LIN {X 0,Y 235.137,Z 262.859,A -85,B 0,C 180,E1 -19747.889,E2 -19747.889} C_VEL
LIN {X 0,Y 235.031,Z 260.731,A -85,B 0,C 180,E1 -19751.62,E2 -19751.62} C_VEL
LIN {X 0,Y 234.887,Z 259.391,A -85,B 0,C 180,E1 -19754.102,E2 -19754.102} C_VEL
LIN {X 0,Y 234.882,Z 259.229,A -85,B 0,C 180,E1 -19758.416,E2 -19758.416} C_VEL
LIN {X 0,Y 234.948,Z 259.217,A -85,B 0,C 180,E1 -19761.084,E2 -19761.084} C_VEL
LIN {X 0,Y 234.953,Z 259.217,A -85,B 0,C 180,E1 -19765.365,E2 -19765.365} C_VEL
LIN {X 0,Y 234.961,Z 259.216,A -85,B 0,C 180,E1 -19770.156,E2 -19770.156} C_VEL
LIN {X 0,Y 234.985,Z 259.213,A -85,B 0,C 180,E1 -19773.792,E2 -19773.792} C_VEL
LIN {X 0,Y 235.002,Z 259.213,A -85,B 0,C 180,E1 -19778.969,E2 -19778.969} C_VEL
LIN {X 0,Y 235.086,Z 259.202,A -85,B 0,C 180,E1 -19783.058,E2 -19783.058} C_VEL
LIN {X 0,Y 235.136,Z 259.195,A -85,B 0,C 180,E1 -19787.923,E2 -19787.923} C_VEL
LIN {X 0,Y 235.381,Z 259.165,A -85,B 0,C 180,E1 -19791.414,E2 -19791.414} C_VEL
LIN {X 0,Y 235.397,Z 259.162,A -85,B 0,C 180,E1 -19793.141,E2 -19793.141} C_VEL
LIN {X 0,Y 235.593,Z 259.138,A -85,B 0,C 180,E1 -19798.29,E2 -19798.29} C_VEL
LIN {X 0,Y 235.586,Z 259.141,A -85,B 0,C 180,E1 -19801.709,E2 -19801.709} C_VEL
LIN {X 0,Y 235.397,Z 259.162,A -85,B 0,C 180,E1 -19806.859,E2 -19806.859} C_VEL
LIN {X 0,Y 235.243,Z 259.182,A -85,B 0,C 180,E1 -19810.326,E2 -19810.326} C_VEL
LIN {X 0,Y 235.103,Z 259.191,A -85,B 0,C 180,E1 -19815.607,E2 -19815.607} C_VEL
LIN {X 0,Y 234.998,Z 259.206,A -85,B 0,C 180,E1 -19819.206,E2 -19819.206} C_VEL
LIN {X 0,Y 234.951,Z 259.218,A -85,B 0,C 180,E1 -19822.884,E2 -19822.884} C_VEL
LIN {X 0,Y 234.96,Z 259.218,A -85,B 0,C 180,E1 -19826.658,E2 -19826.658} C_VEL
LIN {X 0,Y 235.019,Z 259.356,A -85,B 0,C 180,E1 -19829.456,E2 -19829.456} C_VEL
LIN {X 0,Y 235.474,Z 262.099,A -85,B 0,C 180,E1 -19833.317,E2 -19833.317} C_VEL
LIN {X 0,Y 235.891,Z 264.612,A -85,B 0,C 180,E1 -19836.574,E2 -19836.574} C_VEL
LIN {X 0,Y 236.478,Z 268.222,A -85,B 0,C 180,E1 -19840.831,E2 -19840.831} C_VEL
LIN {X 0,Y 237.176,Z 271.785,A -85,B 0,C 180,E1 -19844.674,E2 -19844.674} C_VEL
LIN {X 0,Y 237.723,Z 274.689,A -85,B 0,C 180,E1 -19847.655,E2 -19847.655} C_VEL
LIN {X 0,Y 238.213,Z 278.061,A -85,B 0,C 180,E1 -19850.898,E2 -19850.898} C_VEL
LIN {X 0,Y 237.534,Z 279.156,A -85,B 0,C 180,E1 -19851.795,E2 -19851.795} C_VEL
LIN {X 0,Y 234.488,Z 281.133,A -85,B 0,C 180,E1 -19853.167,E2 -19853.167} C_VEL
LIN {X 0,Y 231.288,Z 283.125,A -85,B 0,C 180,E1 -19854.569,E2 -19854.569} C_VEL
LIN {X 0,Y 230.426,Z 284.271,A -85,B 0,C 180,E1 -19855.504,E2 -19855.504} C_VEL
LIN {X 0,Y 230.39,Z 284.412,A -85,B 0,C 180,E1 -19855.627,E2 -19855.627} C_VEL
LIN {X 0,Y 231.203,Z 287.728,A -85,B 0,C 180,E1 -19855.945,E2 -19855.945} C_VEL
LIN {X 0,Y 234.78,Z 300.694,A -85,B 0,C 180,E1 -19857.465,E2 -19857.465} C_VEL
LIN {X 0,Y 237.057,Z 312.469,A -85,B 0,C 180,E1 -19858.986,E2 -19858.986} C_VEL
LIN {X 0,Y 238.455,Z 324.771,A -85,B 0,C 180,E1 -19860.767,E2 -19860.767} C_VEL
LIN {X 0,Y 238.796,Z 335.33,A -85,B 0,C 180,E1 -19862.512,E2 -19862.512} C_VEL
LIN {X 0,Y 238.284,Z 345.559,A -85,B 0,C 180,E1 -19864.45,E2 -19864.45} C_VEL
LIN {X 0,Y 236.518,Z 352.666,A -85,B 0,C 180,E1 -19865.888,E2 -19865.888} C_VEL
LIN {X 0,Y 234.021,Z 361.179,A -85,B 0,C 180,E1 -19867.954,E2 -19867.954} C_VEL
LIN {X 0,Y 231.65,Z 369.503,A -85,B 0,C 180,E1 -19870.508,E2 -19870.508} C_VEL
LIN {X 0,Y 229.654,Z 376.233,A -85,B 0,C 180,E1 -19873.102,E2 -19873.102} C_VEL
LIN {X 0,Y 227.937,Z 381.62,A -85,B 0,C 180,E1 -19875.723,E2 -19875.723} C_VEL
LIN {X 0,Y 226.866,Z 385.849,A -85,B 0,C 180,E1 -19878.386,E2 -19878.386} C_VEL
LIN {X 0,Y 226.17,Z 389.027,A -85,B 0,C 180,E1 -19881.064,E2 -19881.064} C_VEL
LIN {X 0,Y 225.931,Z 390.624,A -85,B 0,C 180,E1 -19882.855,E2 -19882.855} C_VEL
LIN {X 0,Y 225.839,Z 391.843,A -85,B 0,C 180,E1 -19884.763,E2 -19884.763} C_VEL
LIN {X 0,Y 225.885,Z 392.883,A -85,B 0,C 180,E1 -19888.22,E2 -19888.22} C_VEL
LIN {X 0,Y 225.95,Z 392.842,A -85,B 0,C 180,E1 -19890.003,E2 -19890.003} C_VEL
LIN {X 0,Y 225.909,Z 392.378,A -85,B 0,C 180,E1 -19891.785,E2 -19891.785} C_VEL
LIN {X 0,Y 225.864,Z 391.475,A -85,B 0,C 180,E1 -19893.571,E2 -19893.571} C_VEL
LIN {X 0,Y 225.883,Z 390.17,A -85,B 0,C 180,E1 -19895.358,E2 -19895.358} C_VEL
LIN {X 0,Y 226.081,Z 387.399,A -85,B 0,C 180,E1 -19898.044,E2 -19898.044} C_VEL
LIN {X 0,Y 226.596,Z 383.592,A -85,B 0,C 180,E1 -19900.727,E2 -19900.727} C_VEL
LIN {X 0,Y 227.465,Z 378.65,A -85,B 0,C 180,E1 -19903.401,E2 -19903.401} C_VEL
LIN {X 0,Y 228.927,Z 372.442,A -85,B 0,C 180,E1 -19906.042,E2 -19906.042} C_VEL
LIN {X 0,Y 230.66,Z 364.83,A -85,B 0,C 180,E1 -19908.623,E2 -19908.623} C_VEL
LIN {X 0,Y 232.391,Z 356.97,A -85,B 0,C 180,E1 -19910.771,E2 -19910.771} C_VEL
LIN {X 0,Y 234.323,Z 348.211,A -85,B 0,C 180,E1 -19912.718,E2 -19912.718} C_VEL
LIN {X 0,Y 235.388,Z 342.642,A -85,B 0,C 180,E1 -19913.773,E2 -19913.773} C_VEL
LIN {X 0,Y 235.357,Z 331.167,A -85,B 0,C 180,E1 -19915.788,E2 -19915.788} C_VEL
LIN {X 0,Y 234.896,Z 319.818,A -85,B 0,C 180,E1 -19917.434,E2 -19917.434} C_VEL
LIN {X 0,Y 233.577,Z 307.331,A -85,B 0,C 180,E1 -19918.943,E2 -19918.943} C_VEL
LIN {X 0,Y 231.149,Z 294.067,A -85,B 0,C 180,E1 -19920.296,E2 -19920.296} C_VEL
LIN {X 0,Y 229.071,Z 284.971,A -85,B 0,C 180,E1 -19921.1,E2 -19921.1} C_VEL
LIN {X 0,Y 230.358,Z 279.833,A -85,B 0,C 180,E1 -19925.43,E2 -19925.43} C_VEL
LIN {X 0,Y 230.728,Z 277.284,A -85,B 0,C 180,E1 -19927.631,E2 -19927.631} C_VEL
LIN {X 0,Y 230.496,Z 274.331,A -85,B 0,C 180,E1 -19930.335,E2 -19930.335} C_VEL
LIN {X 0,Y 229.629,Z 269.831,A -85,B 0,C 180,E1 -19934.747,E2 -19934.747} C_VEL
LIN {X 0,Y 228.975,Z 266.081,A -85,B 0,C 180,E1 -19938.707,E2 -19938.707} C_VEL
LIN {X 0,Y 228.326,Z 262.168,A -85,B 0,C 180,E1 -19943.162,E2 -19943.162} C_VEL
LIN {X 0,Y 227.892,Z 260.098,A -85,B 0,C 180,E1 -19945.749,E2 -19945.749} C_VEL
LIN {X 0,Y 227.884,Z 260.098,A -85,B 0,C 180,E1 -19950.433,E2 -19950.433} C_VEL
LIN {X 0,Y 227.912,Z 260.095,A -85,B 0,C 180,E1 -19954.424,E2 -19954.424} C_VEL
LIN {X 0,Y 227.955,Z 260.091,A -85,B 0,C 180,E1 -19958.286,E2 -19958.286} C_VEL
LIN {X 0,Y 227.998,Z 260.084,A -85,B 0,C 180,E1 -19962.864,E2 -19962.864} C_VEL
LIN {X 0,Y 228.051,Z 260.08,A -85,B 0,C 180,E1 -19967.542,E2 -19967.542} C_VEL
LIN {X 0,Y 228.259,Z 260.053,A -85,B 0,C 180,E1 -19971.144,E2 -19971.144} C_VEL
LIN {X 0,Y 228.325,Z 260.041,A -85,B 0,C 180,E1 -19972.928,E2 -19972.928} C_VEL
LIN {X 0,Y 228.562,Z 260.014,A -85,B 0,C 180,E1 -19978.238,E2 -19978.238} C_VEL
LIN {X 0,Y 228.547,Z 260.017,A -85,B 0,C 180,E1 -19981.762,E2 -19981.762} C_VEL
LIN {X 0,Y 228.309,Z 260.046,A -85,B 0,C 180,E1 -19987.073,E2 -19987.073} C_VEL
LIN {X 0,Y 228.151,Z 260.061,A -85,B 0,C 180,E1 -19990.651,E2 -19990.651} C_VEL
LIN {X 0,Y 228.046,Z 260.074,A -85,B 0,C 180,E1 -19994.274,E2 -19994.274} C_VEL
LIN {X 0,Y 227.962,Z 260.087,A -85,B 0,C 180,E1 -19997.957,E2 -19997.957} C_VEL
LIN {X 0,Y 227.913,Z 260.095,A -85,B 0,C 180,E1 -20002.312,E2 -20002.312} C_VEL
LIN {X 0,Y 227.91,Z 260.096,A -85,B 0,C 180,E1 -20006.581,E2 -20006.581} C_VEL
LIN {X 0,Y 227.878,Z 260.098,A -85,B 0,C 180,E1 -20010.278,E2 -20010.278} C_VEL
LIN {X 0,Y 227.885,Z 260.095,A -85,B 0,C 180,E1 -20013.72,E2 -20013.72} C_VEL
LIN {X 0,Y 227.852,Z 260.102,A -85,B 0,C 180,E1 -20018.09,E2 -20018.09} C_VEL
LIN {X 0,Y 227.813,Z 260.106,A -85,B 0,C 180,E1 -20022.742,E2 -20022.742} C_VEL
LIN {X 0,Y 227.797,Z 260.109,A -85,B 0,C 180,E1 -20027.251,E2 -20027.251} C_VEL
LIN {X 0,Y 227.844,Z 260.104,A -85,B 0,C 180,E1 -20031.906,E2 -20031.906} C_VEL
LIN {X 0,Y 227.82,Z 260.105,A -85,B 0,C 180,E1 -20036.267,E2 -20036.267} C_VEL
LIN {X 0,Y 227.682,Z 260.118,A -85,B 0,C 180,E1 -20038.346,E2 -20038.346} C_VEL
LIN {X 0,Y 227.603,Z 260.825,A -85,B 0,C 180,E1 -20040.39,E2 -20040.39} C_VEL
LIN {X 0,Y 227.534,Z 262.75,A -85,B 0,C 180,E1 -20043.143,E2 -20043.143} C_VEL
LIN {X 0,Y 228.668,Z 265.801,A -85,B 0,C 180,E1 -20043.474,E2 -20043.474} C_VEL
LIN {X 0,Y 232.897,Z 277.354,A -85,B 0,C 180,E1 -20044.864,E2 -20044.864} C_VEL
LIN {X 0,Y 235.978,Z 288.099,A -85,B 0,C 180,E1 -20046.305,E2 -20046.305} C_VEL
LIN {X 0,Y 238.279,Z 299.414,A -85,B 0,C 180,E1 -20048.005,E2 -20048.005} C_VEL
LIN {X 0,Y 239.076,Z 305.229,A -85,B 0,C 180,E1 -20048.976,E2 -20048.976} C_VEL
LIN {X 0,Y 237.375,Z 315.143,A -85,B 0,C 180,E1 -20050.542,E2 -20050.542} C_VEL
LIN {X 0,Y 235.171,Z 325.68,A -85,B 0,C 180,E1 -20052.609,E2 -20052.609} C_VEL
LIN {X 0,Y 233.368,Z 333.508,A -85,B 0,C 180,E1 -20054.516,E2 -20054.516} C_VEL
LIN {X 0,Y 231.558,Z 341.294,A -85,B 0,C 180,E1 -20056.84,E2 -20056.84} C_VEL
LIN {X 0,Y 229.715,Z 348.233,A -85,B 0,C 180,E1 -20059.42,E2 -20059.42} C_VEL
LIN {X 0,Y 228.841,Z 352.047,A -85,B 0,C 180,E1 -20061.164,E2 -20061.164} C_VEL
LIN {X 0,Y 227.754,Z 356.785,A -85,B 0,C 180,E1 -20063.797,E2 -20063.797} C_VEL
LIN {X 0,Y 226.813,Z 360.44,A -85,B 0,C 180,E1 -20066.444,E2 -20066.444} C_VEL
LIN {X 0,Y 226.45,Z 362.325,A -85,B 0,C 180,E1 -20068.219,E2 -20068.219} C_VEL
LIN {X 0,Y 226.197,Z 363.78,A -85,B 0,C 180,E1 -20069.997,E2 -20069.997} C_VEL
LIN {X 0,Y 226.135,Z 365.446,A -85,B 0,C 180,E1 -20073.561,E2 -20073.561} C_VEL
LIN {X 0,Y 226.283,Z 365.678,A -85,B 0,C 180,E1 -20076.342,E2 -20076.342} C_VEL
LIN {X 0,Y 226.504,Z 365.058,A -85,B 0,C 180,E1 -20078.922,E2 -20078.922} C_VEL
LIN {X 0,Y 227.34,Z 362.821,A -85,B 0,C 180,E1 -20082.495,E2 -20082.495} C_VEL
LIN {X 0,Y 228.402,Z 360.02,A -85,B 0,C 180,E1 -20085.159,E2 -20085.159} C_VEL
LIN {X 0,Y 229.798,Z 356.193,A -85,B 0,C 180,E1 -20087.806,E2 -20087.806} C_VEL
LIN {X 0,Y 231.579,Z 351.225,A -85,B 0,C 180,E1 -20090.424,E2 -20090.424} C_VEL
LIN {X 0,Y 233.827,Z 344.95,A -85,B 0,C 180,E1 -20092.997,E2 -20092.997} C_VEL
LIN {X 0,Y 236.355,Z 337.063,A -85,B 0,C 180,E1 -20095.538,E2 -20095.538} C_VEL
LIN {X 0,Y 238.723,Z 329.001,A -85,B 0,C 180,E1 -20097.622,E2 -20097.622} C_VEL
LIN {X 0,Y 241.366,Z 319.137,A -85,B 0,C 180,E1 -20099.667,E2 -20099.667} C_VEL
LIN {X 0,Y 243.113,Z 311.993,A -85,B 0,C 180,E1 -20100.869,E2 -20100.869} C_VEL
LIN {X 0,Y 241.935,Z 302.961,A -85,B 0,C 180,E1 -20102.602,E2 -20102.602} C_VEL
LIN {X 0,Y 239.585,Z 292.859,A -85,B 0,C 180,E1 -20104.409,E2 -20104.409} C_VEL
LIN {X 0,Y 235.756,Z 280.778,A -85,B 0,C 180,E1 -20106.4,E2 -20106.4} C_VEL
LIN {X 0,Y 231.266,Z 270.388,A -85,B 0,C 180,E1 -20108.062,E2 -20108.062} C_VEL
LIN {X 0,Y 229.347,Z 266.528,A -85,B 0,C 180,E1 -20108.669,E2 -20108.669} C_VEL
LIN {X 0,Y 228.101,Z 263.373,A -85,B 0,C 180,E1 -20109.132,E2 -20109.132} C_VEL
LIN {X 0,Y 227.97,Z 261.447,A -85,B 0,C 180,E1 -20112.702,E2 -20112.702} C_VEL
LIN {X 0,Y 227.819,Z 260.161,A -85,B 0,C 180,E1 -20115.192,E2 -20115.192} C_VEL
LIN {X 0,Y 227.825,Z 260.106,A -85,B 0,C 180,E1 -20119.623,E2 -20119.623} C_VEL
LIN {X 0,Y 227.892,Z 260.096,A -85,B 0,C 180,E1 -20124.13,E2 -20124.13} C_VEL
LIN {X 0,Y 227.864,Z 260.099,A -85,B 0,C 180,E1 -20128.376,E2 -20128.376} C_VEL
LIN {X 0,Y 227.877,Z 260.093,A -85,B 0,C 180,E1 -20132.443,E2 -20132.443} C_VEL
LIN {X 0,Y 227.905,Z 260.097,A -85,B 0,C 180,E1 -20136.366,E2 -20136.366} C_VEL
LIN {X 0,Y 227.933,Z 260.092,A -85,B 0,C 180,E1 -20140.173,E2 -20140.173} C_VEL
LIN {X 0,Y 228.048,Z 260.077,A -85,B 0,C 180,E1 -20143.897,E2 -20143.897} C_VEL
LIN {X 0,Y 228.161,Z 260.066,A -85,B 0,C 180,E1 -20149.349,E2 -20149.349} C_VEL
LIN {X 0,Y 228.349,Z 260.04,A -85,B 0,C 180,E1 -20152.928,E2 -20152.928} C_VEL
LIN {X 0,Y 228.553,Z 260.015,A -85,B 0,C 180,E1 -20158.238,E2 -20158.238} C_VEL
LIN {X 0,Y 228.545,Z 260.018,A -85,B 0,C 180,E1 -20161.762,E2 -20161.762} C_VEL
LIN {X 0,Y 228.349,Z 260.04,A -85,B 0,C 180,E1 -20167.071,E2 -20167.071} C_VEL
LIN {X 0,Y 228.161,Z 260.063,A -85,B 0,C 180,E1 -20170.65,E2 -20170.65} C_VEL
LIN {X 0,Y 228.047,Z 260.071,A -85,B 0,C 180,E1 -20176.103,E2 -20176.103} C_VEL
LIN {X 0,Y 227.932,Z 260.088,A -85,B 0,C 180,E1 -20179.826,E2 -20179.826} C_VEL
LIN {X 0,Y 227.904,Z 260.098,A -85,B 0,C 180,E1 -20183.634,E2 -20183.634} C_VEL
LIN {X 0,Y 227.891,Z 260.132,A -85,B 0,C 180,E1 -20188.054,E2 -20188.054} C_VEL
LIN {X 0,Y 228.311,Z 262.418,A -85,B 0,C 180,E1 -20191.554,E2 -20191.554} C_VEL
LIN {X 0,Y 228.812,Z 265.456,A -85,B 0,C 180,E1 -20195.703,E2 -20195.703} C_VEL
LIN {X 0,Y 229.4,Z 268.969,A -85,B 0,C 180,E1 -20200.043,E2 -20200.043} C_VEL
LIN {X 0,Y 229.887,Z 271.346,A -85,B 0,C 180,E1 -20202.805,E2 -20202.805} C_VEL
LIN {X 0,Y 230.615,Z 275.277,A -85,B 0,C 180,E1 -20207.004,E2 -20207.004} C_VEL
LIN {X 0,Y 231.178,Z 278.574,A -85,B 0,C 180,E1 -20210.33,E2 -20210.33} C_VEL
LIN {X 0,Y 231.238,Z 280.951,A -85,B 0,C 180,E1 -20212.569,E2 -20212.569} C_VEL
LIN {X 0,Y 230.426,Z 284.271,A -85,B 0,C 180,E1 -20215.504,E2 -20215.504} C_VEL
LIN {X 0,Y 231.228,Z 285.071,A -85,B 0,C 180,E1 -20215.808,E2 -20215.808} C_VEL
LIN {X 0,Y 233.342,Z 287.602,A -85,B 0,C 180,E1 -20216.31,E2 -20216.31} C_VEL
LIN {X 0,Y 234.902,Z 290.926,A -85,B 0,C 180,E1 -20216.743,E2 -20216.743} C_VEL
LIN {X 0,Y 235.443,Z 294.756,A -85,B 0,C 180,E1 -20217.111,E2 -20217.111} C_VEL
LIN {X 0,Y 235.158,Z 299.092,A -85,B 0,C 180,E1 -20217.313,E2 -20217.313} C_VEL
LIN {X 0,Y 232.838,Z 305.681,A -85,B 0,C 180,E1 -20217.51,E2 -20217.51} C_VEL
LIN {X 0,Y 230.998,Z 310.912,A -85,B 0,C 180,E1 -20217.847,E2 -20217.847} C_VEL
LIN {X 0,Y 230.809,Z 313.949,A -85,B 0,C 180,E1 -20218.202,E2 -20218.202} C_VEL
LIN {X 0,Y 232.06,Z 326.581,A -85,B 0,C 180,E1 -20220.164,E2 -20220.164} C_VEL
LIN {X 0,Y 232.24,Z 337.478,A -85,B 0,C 180,E1 -20222.09,E2 -20222.09} C_VEL
LIN {X 0,Y 231.473,Z 347.568,A -85,B 0,C 180,E1 -20224.125,E2 -20224.125} C_VEL
LIN {X 0,Y 228.928,Z 356.07,A -85,B 0,C 180,E1 -20226.001,E2 -20226.001} C_VEL
LIN {X 0,Y 226.109,Z 365.279,A -85,B 0,C 180,E1 -20228.57,E2 -20228.57} C_VEL
LIN {X 0,Y 223.823,Z 372.77,A -85,B 0,C 180,E1 -20231.228,E2 -20231.228} C_VEL
LIN {X 0,Y 221.593,Z 379.667,A -85,B 0,C 180,E1 -20234.363,E2 -20234.363} C_VEL
LIN {X 0,Y 220.177,Z 384.236,A -85,B 0,C 180,E1 -20237.092,E2 -20237.092} C_VEL
LIN {X 0,Y 219.588,Z 386.662,A -85,B 0,C 180,E1 -20238.931,E2 -20238.931} C_VEL
LIN {X 0,Y 219.137,Z 388.658,A -85,B 0,C 180,E1 -20240.775,E2 -20240.775} C_VEL
LIN {X 0,Y 218.856,Z 390.243,A -85,B 0,C 180,E1 -20242.623,E2 -20242.623} C_VEL
LIN {X 0,Y 218.74,Z 391.573,A -85,B 0,C 180,E1 -20244.884,E2 -20244.884} C_VEL
LIN {X 0,Y 218.815,Z 392.462,A -85,B 0,C 180,E1 -20248.162,E2 -20248.162} C_VEL
LIN {X 0,Y 218.878,Z 392.411,A -85,B 0,C 180,E1 -20250.003,E2 -20250.003} C_VEL
LIN {X 0,Y 218.838,Z 391.925,A -85,B 0,C 180,E1 -20251.843,E2 -20251.843} C_VEL
LIN {X 0,Y 218.784,Z 389.925,A -85,B 0,C 180,E1 -20255.244,E2 -20255.244} C_VEL
LIN {X 0,Y 219.043,Z 386.899,A -85,B 0,C 180,E1 -20258.304,E2 -20258.304} C_VEL
LIN {X 0,Y 219.596,Z 383.067,A -85,B 0,C 180,E1 -20261.074,E2 -20261.074} C_VEL
LIN {X 0,Y 220.533,Z 378.098,A -85,B 0,C 180,E1 -20263.831,E2 -20263.831} C_VEL
LIN {X 0,Y 222.031,Z 371.857,A -85,B 0,C 180,E1 -20266.554,E2 -20266.554} C_VEL
LIN {X 0,Y 223.782,Z 364.6,A -85,B 0,C 180,E1 -20269.085,E2 -20269.085} C_VEL
LIN {X 0,Y 225.736,Z 356.116,A -85,B 0,C 180,E1 -20271.461,E2 -20271.461} C_VEL
LIN {X 0,Y 227.976,Z 346.407,A -85,B 0,C 180,E1 -20273.628,E2 -20273.628} C_VEL
LIN {X 0,Y 228.546,Z 343.068,A -85,B 0,C 180,E1 -20274.289,E2 -20274.289} C_VEL
LIN {X 0,Y 228.641,Z 330.99,A -85,B 0,C 180,E1 -20276.49,E2 -20276.49} C_VEL
LIN {X 0,Y 228.27,Z 320.835,A -85,B 0,C 180,E1 -20278.033,E2 -20278.033} C_VEL
LIN {X 0,Y 226.993,Z 307.895,A -85,B 0,C 180,E1 -20279.698,E2 -20279.698} C_VEL
LIN {X 0,Y 224.528,Z 294.296,A -85,B 0,C 180,E1 -20281.164,E2 -20281.164} C_VEL
LIN {X 0,Y 222.295,Z 285.273,A -85,B 0,C 180,E1 -20282.009,E2 -20282.009} C_VEL
LIN {X 0,Y 222.241,Z 284.55,A -85,B 0,C 180,E1 -20282.072,E2 -20282.072} C_VEL
LIN {X 0,Y 223.143,Z 281.169,A -85,B 0,C 180,E1 -20285.027,E2 -20285.027} C_VEL
LIN {X 0,Y 223.579,Z 279.31,A -85,B 0,C 180,E1 -20286.676,E2 -20286.676} C_VEL
LIN {X 0,Y 223.665,Z 276.847,A -85,B 0,C 180,E1 -20288.938,E2 -20288.938} C_VEL
LIN {X 0,Y 223.07,Z 273.235,A -85,B 0,C 180,E1 -20292.46,E2 -20292.46} C_VEL
LIN {X 0,Y 222.319,Z 269.265,A -85,B 0,C 180,E1 -20296.646,E2 -20296.646} C_VEL
LIN {X 0,Y 221.662,Z 265.72,A -85,B 0,C 180,E1 -20300.645,E2 -20300.645} C_VEL
LIN {X 0,Y 221.405,Z 263.799,A -85,B 0,C 180,E1 -20302.907,E2 -20302.907} C_VEL
LIN {X 0,Y 220.845,Z 260.976,A -85,B 0,C 180,E1 -20306.521,E2 -20306.521} C_VEL
LIN {X 0,Y 220.842,Z 260.975,A -85,B 0,C 180,E1 -20309.391,E2 -20309.391} C_VEL
LIN {X 0,Y 220.884,Z 260.969,A -85,B 0,C 180,E1 -20313.548,E2 -20313.548} C_VEL
LIN {X 0,Y 220.877,Z 260.971,A -85,B 0,C 180,E1 -20317.553,E2 -20317.553} C_VEL
LIN {X 0,Y 220.936,Z 260.965,A -85,B 0,C 180,E1 -20322.62,E2 -20322.62} C_VEL
LIN {X 0,Y 220.984,Z 260.959,A -85,B 0,C 180,E1 -20327.137,E2 -20327.137} C_VEL
LIN {X 0,Y 221.196,Z 260.932,A -85,B 0,C 180,E1 -20330.859,E2 -20330.859} C_VEL
LIN {X 0,Y 221.259,Z 260.921,A -85,B 0,C 180,E1 -20332.701,E2 -20332.701} C_VEL
LIN {X 0,Y 221.52,Z 260.891,A -85,B 0,C 180,E1 -20338.182,E2 -20338.182} C_VEL
LIN {X 0,Y 221.481,Z 260.897,A -85,B 0,C 180,E1 -20341.819,E2 -20341.819} C_VEL
LIN {X 0,Y 221.247,Z 260.927,A -85,B 0,C 180,E1 -20347.3,E2 -20347.3} C_VEL
LIN {X 0,Y 221.072,Z 260.945,A -85,B 0,C 180,E1 -20350.996,E2 -20350.996} C_VEL
LIN {X 0,Y 220.988,Z 260.957,A -85,B 0,C 180,E1 -20356.632,E2 -20356.632} C_VEL
LIN {X 0,Y 220.883,Z 260.966,A -85,B 0,C 180,E1 -20360.487,E2 -20360.487} C_VEL
LIN {X 0,Y 220.806,Z 260.977,A -85,B 0,C 180,E1 -20364.443,E2 -20364.443} C_VEL
LIN {X 0,Y 220.804,Z 260.979,A -85,B 0,C 180,E1 -20368.519,E2 -20368.519} C_VEL
LIN {X 0,Y 220.82,Z 260.976,A -85,B 0,C 180,E1 -20372.756,E2 -20372.756} C_VEL
LIN {X 0,Y 220.819,Z 260.977,A -85,B 0,C 180,E1 -20377.277,E2 -20377.277} C_VEL
LIN {X 0,Y 220.803,Z 260.98,A -85,B 0,C 180,E1 -20380.187,E2 -20380.187} C_VEL
LIN {X 0,Y 220.773,Z 260.985,A -85,B 0,C 180,E1 -20384.455,E2 -20384.455} C_VEL
LIN {X 0,Y 220.756,Z 260.987,A -85,B 0,C 180,E1 -20388.041,E2 -20388.041} C_VEL
LIN {X 0,Y 220.832,Z 260.977,A -85,B 0,C 180,E1 -20392.791,E2 -20392.791} C_VEL
LIN {X 0,Y 220.693,Z 260.991,A -85,B 0,C 180,E1 -20397.22,E2 -20397.22} C_VEL
LIN {X 0,Y 220.612,Z 261.328,A -85,B 0,C 180,E1 -20399.353,E2 -20399.353} C_VEL
LIN {X 0,Y 220.493,Z 263.082,A -85,B 0,C 180,E1 -20402.107,E2 -20402.107} C_VEL
LIN {X 0,Y 221.673,Z 266.22,A -85,B 0,C 180,E1 -20402.467,E2 -20402.467} C_VEL
LIN {X 0,Y 225.988,Z 277.513,A -85,B 0,C 180,E1 -20403.922,E2 -20403.922} C_VEL
LIN {X 0,Y 229.395,Z 289.296,A -85,B 0,C 180,E1 -20405.582,E2 -20405.582} C_VEL
LIN {X 0,Y 231.459,Z 299.28,A -85,B 0,C 180,E1 -20407.153,E2 -20407.153} C_VEL
LIN {X 0,Y 232.418,Z 306.206,A -85,B 0,C 180,E1 -20408.355,E2 -20408.355} C_VEL
LIN {X 0,Y 230.498,Z 317.12,A -85,B 0,C 180,E1 -20410.169,E2 -20410.169} C_VEL
LIN {X 0,Y 228.461,Z 326.428,A -85,B 0,C 180,E1 -20412.081,E2 -20412.081} C_VEL
LIN {X 0,Y 226.534,Z 334.432,A -85,B 0,C 180,E1 -20414.102,E2 -20414.102} C_VEL
LIN {X 0,Y 224.685,Z 341.939,A -85,B 0,C 180,E1 -20416.43,E2 -20416.43} C_VEL
LIN {X 0,Y 222.774,Z 348.825,A -85,B 0,C 180,E1 -20419.086,E2 -20419.086} C_VEL
LIN {X 0,Y 221.852,Z 352.623,A -85,B 0,C 180,E1 -20420.884,E2 -20420.884} C_VEL
LIN {X 0,Y 220.739,Z 357.328,A -85,B 0,C 180,E1 -20423.599,E2 -20423.599} C_VEL
LIN {X 0,Y 219.745,Z 360.955,A -85,B 0,C 180,E1 -20426.33,E2 -20426.33} C_VEL
LIN {X 0,Y 219.368,Z 362.826,A -85,B 0,C 180,E1 -20428.161,E2 -20428.161} C_VEL
LIN {X 0,Y 219.114,Z 364.253,A -85,B 0,C 180,E1 -20429.997,E2 -20429.997} C_VEL
LIN {X 0,Y 219.074,Z 365.892,A -85,B 0,C 180,E1 -20433.676,E2 -20433.676} C_VEL
LIN {X 0,Y 219.209,Z 366.115,A -85,B 0,C 180,E1 -20436.337,E2 -20436.337} C_VEL
LIN {X 0,Y 219.482,Z 365.452,A -85,B 0,C 180,E1 -20439.21,E2 -20439.21} C_VEL
LIN {X 0,Y 220.382,Z 363.19,A -85,B 0,C 180,E1 -20442.896,E2 -20442.896} C_VEL
LIN {X 0,Y 221.524,Z 360.361,A -85,B 0,C 180,E1 -20445.642,E2 -20445.642} C_VEL
LIN {X 0,Y 223.003,Z 356.503,A -85,B 0,C 180,E1 -20448.367,E2 -20448.367} C_VEL
LIN {X 0,Y 224.891,Z 351.503,A -85,B 0,C 180,E1 -20451.059,E2 -20451.059} C_VEL
LIN {X 0,Y 227.252,Z 345.178,A -85,B 0,C 180,E1 -20453.703,E2 -20453.703} C_VEL
LIN {X 0,Y 229.943,Z 337.243,A -85,B 0,C 180,E1 -20456.304,E2 -20456.304} C_VEL
LIN {X 0,Y 232.39,Z 329.188,A -85,B 0,C 180,E1 -20458.426,E2 -20458.426} C_VEL
LIN {X 0,Y 235.202,Z 319.207,A -85,B 0,C 180,E1 -20460.526,E2 -20460.526} C_VEL
LIN {X 0,Y 236.713,Z 313.282,A -85,B 0,C 180,E1 -20461.55,E2 -20461.55} C_VEL
LIN {X 0,Y 235.255,Z 303.035,A -85,B 0,C 180,E1 -20463.619,E2 -20463.619} C_VEL
LIN {X 0,Y 232.587,Z 292.077,A -85,B 0,C 180,E1 -20465.664,E2 -20465.664} C_VEL
LIN {X 0,Y 229.118,Z 281.59,A -85,B 0,C 180,E1 -20467.495,E2 -20467.495} C_VEL
LIN {X 0,Y 224.613,Z 271.275,A -85,B 0,C 180,E1 -20469.262,E2 -20469.262} C_VEL
LIN {X 0,Y 222.301,Z 267.032,A -85,B 0,C 180,E1 -20470.018,E2 -20470.018} C_VEL
LIN {X 0,Y 221.095,Z 263.875,A -85,B 0,C 180,E1 -20470.509,E2 -20470.509} C_VEL
LIN {X 0,Y 220.878,Z 261.88,A -85,B 0,C 180,E1 -20474.423,E2 -20474.423} C_VEL
LIN {X 0,Y 220.755,Z 260.987,A -85,B 0,C 180,E1 -20477.069,E2 -20477.069} C_VEL
LIN {X 0,Y 220.802,Z 260.981,A -85,B 0,C 180,E1 -20480.462,E2 -20480.462} C_VEL
LIN {X 0,Y 220.824,Z 260.977,A -85,B 0,C 180,E1 -20482.792,E2 -20482.792} C_VEL
LIN {X 0,Y 220.816,Z 260.979,A -85,B 0,C 180,E1 -20487.243,E2 -20487.243} C_VEL
LIN {X 0,Y 220.828,Z 260.977,A -85,B 0,C 180,E1 -20491.485,E2 -20491.485} C_VEL
LIN {X 0,Y 220.858,Z 260.973,A -85,B 0,C 180,E1 -20495.564,E2 -20495.564} C_VEL
LIN {X 0,Y 220.883,Z 260.97,A -85,B 0,C 180,E1 -20499.513,E2 -20499.513} C_VEL
LIN {X 0,Y 221.007,Z 260.956,A -85,B 0,C 180,E1 -20503.369,E2 -20503.369} C_VEL
LIN {X 0,Y 221.107,Z 260.942,A -85,B 0,C 180,E1 -20509.005,E2 -20509.005} C_VEL
LIN {X 0,Y 221.302,Z 260.918,A -85,B 0,C 180,E1 -20512.702,E2 -20512.702} C_VEL
LIN {X 0,Y 221.511,Z 260.892,A -85,B 0,C 180,E1 -20518.182,E2 -20518.182} C_VEL
LIN {X 0,Y 221.503,Z 260.894,A -85,B 0,C 180,E1 -20521.818,E2 -20521.818} C_VEL
LIN {X 0,Y 221.302,Z 260.919,A -85,B 0,C 180,E1 -20527.298,E2 -20527.298} C_VEL
LIN {X 0,Y 221.106,Z 260.941,A -85,B 0,C 180,E1 -20530.994,E2 -20530.994} C_VEL
LIN {X 0,Y 221.006,Z 260.951,A -85,B 0,C 180,E1 -20536.63,E2 -20536.63} C_VEL
LIN {X 0,Y 220.882,Z 260.971,A -85,B 0,C 180,E1 -20540.487,E2 -20540.487} C_VEL
LIN {X 0,Y 220.858,Z 260.974,A -85,B 0,C 180,E1 -20544.436,E2 -20544.436} C_VEL
LIN {X 0,Y 220.883,Z 261.173,A -85,B 0,C 180,E1 -20547.021,E2 -20547.021} C_VEL
LIN {X 0,Y 221.338,Z 263.628,A -85,B 0,C 180,E1 -20550.989,E2 -20550.989} C_VEL
LIN {X 0,Y 221.745,Z 266.289,A -85,B 0,C 180,E1 -20554.785,E2 -20554.785} C_VEL
LIN {X 0,Y 222.314,Z 269.722,A -85,B 0,C 180,E1 -20559.217,E2 -20559.217} C_VEL
LIN {X 0,Y 223.065,Z 273.646,A -85,B 0,C 180,E1 -20563.88,E2 -20563.88} C_VEL
LIN {X 0,Y 223.726,Z 277.015,A -85,B 0,C 180,E1 -20567.568,E2 -20567.568} C_VEL
LIN {X 0,Y 224.14,Z 279.415,A -85,B 0,C 180,E1 -20570.053,E2 -20570.053} C_VEL
LIN {X 0,Y 224.194,Z 280.983,A -85,B 0,C 180,E1 -20571.6,E2 -20571.6} C_VEL
LIN {X 0,Y 223.718,Z 283.921,A -85,B 0,C 180,E1 -20574.346,E2 -20574.346} C_VEL
LIN {X 0,Y 224.62,Z 287.385,A -85,B 0,C 180,E1 -20574.724,E2 -20574.724} C_VEL
LIN {X 0,Y 228.325,Z 300.717,A -85,B 0,C 180,E1 -20576.388,E2 -20576.388} C_VEL
LIN {X 0,Y 230.718,Z 313.271,A -85,B 0,C 180,E1 -20578.103,E2 -20578.103} C_VEL
LIN {X 0,Y 230.809,Z 313.949,A -85,B 0,C 180,E1 -20578.202,E2 -20578.202} C_VEL
LIN {X 0,Y 230.84,Z 319.234,A -85,B 0,C 180,E1 -20578.893,E2 -20578.893} C_VEL
LIN {X 0,Y 229.832,Z 324.594,A -85,B 0,C 180,E1 -20579.526,E2 -20579.526} C_VEL
LIN {X 0,Y 226.777,Z 334.876,A -85,B 0,C 180,E1 -20580.86,E2 -20580.86} C_VEL
LIN {X 0,Y 225.716,Z 339.706,A -85,B 0,C 180,E1 -20581.682,E2 -20581.682} C_VEL
LIN {X 0,Y 225.562,Z 341.232,A -85,B 0,C 180,E1 -20581.989,E2 -20581.989} C_VEL
LIN {X 0,Y 224.797,Z 348.431,A -85,B 0,C 180,E1 -20583.547,E2 -20583.547} C_VEL
LIN {X 0,Y 221.905,Z 357.53,A -85,B 0,C 180,E1 -20585.69,E2 -20585.69} C_VEL
LIN {X 0,Y 219.017,Z 366.433,A -85,B 0,C 180,E1 -20588.349,E2 -20588.349} C_VEL
LIN {X 0,Y 216.692,Z 373.605,A -85,B 0,C 180,E1 -20591.078,E2 -20591.078} C_VEL
LIN {X 0,Y 214.732,Z 379.346,A -85,B 0,C 180,E1 -20593.85,E2 -20593.85} C_VEL
LIN {X 0,Y 213.213,Z 383.89,A -85,B 0,C 180,E1 -20596.662,E2 -20596.662} C_VEL
LIN {X 0,Y 212.573,Z 386.303,A -85,B 0,C 180,E1 -20598.561,E2 -20598.561} C_VEL
LIN {X 0,Y 212.098,Z 388.288,A -85,B 0,C 180,E1 -20600.466,E2 -20600.466} C_VEL
LIN {X 0,Y 211.808,Z 389.861,A -85,B 0,C 180,E1 -20602.376,E2 -20602.376} C_VEL
LIN {X 0,Y 211.643,Z 391.302,A -85,B 0,C 180,E1 -20605.007,E2 -20605.007} C_VEL
LIN {X 0,Y 211.745,Z 392.041,A -85,B 0,C 180,E1 -20608.101,E2 -20608.101} C_VEL
LIN {X 0,Y 211.808,Z 391.979,A -85,B 0,C 180,E1 -20610.003,E2 -20610.003} C_VEL
LIN {X 0,Y 211.769,Z 391.472,A -85,B 0,C 180,E1 -20611.905,E2 -20611.905} C_VEL
LIN {X 0,Y 211.697,Z 389.651,A -85,B 0,C 180,E1 -20615.157,E2 -20615.157} C_VEL
LIN {X 0,Y 211.978,Z 386.397,A -85,B 0,C 180,E1 -20618.583,E2 -20618.583} C_VEL
LIN {X 0,Y 212.574,Z 382.538,A -85,B 0,C 180,E1 -20621.444,E2 -20621.444} C_VEL
LIN {X 0,Y 213.624,Z 377.546,A -85,B 0,C 180,E1 -20624.288,E2 -20624.288} C_VEL
LIN {X 0,Y 215.149,Z 371.271,A -85,B 0,C 180,E1 -20627.1,E2 -20627.1} C_VEL
LIN {X 0,Y 216.845,Z 364.732,A -85,B 0,C 180,E1 -20629.452,E2 -20629.452} C_VEL
LIN {X 0,Y 218.675,Z 357.164,A -85,B 0,C 180,E1 -20631.694,E2 -20631.694} C_VEL
LIN {X 0,Y 220.984,Z 347.844,A -85,B 0,C 180,E1 -20633.925,E2 -20633.925} C_VEL
LIN {X 0,Y 221.719,Z 343.485,A -85,B 0,C 180,E1 -20634.837,E2 -20634.837} C_VEL
LIN {X 0,Y 221.941,Z 333.136,A -85,B 0,C 180,E1 -20636.836,E2 -20636.836} C_VEL
LIN {X 0,Y 221.712,Z 322.612,A -85,B 0,C 180,E1 -20638.552,E2 -20638.552} C_VEL
LIN {X 0,Y 220.683,Z 310.326,A -85,B 0,C 180,E1 -20640.25,E2 -20640.25} C_VEL
LIN {X 0,Y 218.5,Z 297.045,A -85,B 0,C 180,E1 -20641.822,E2 -20641.822} C_VEL
LIN {X 0,Y 215.476,Z 284.073,A -85,B 0,C 180,E1 -20643.169,E2 -20643.169} C_VEL
LIN {X 0,Y 216.551,Z 279.962,A -85,B 0,C 180,E1 -20646.902,E2 -20646.902} C_VEL
LIN {X 0,Y 216.653,Z 277.913,A -85,B 0,C 180,E1 -20648.874,E2 -20648.874} C_VEL
LIN {X 0,Y 215.928,Z 273.709,A -85,B 0,C 180,E1 -20653.122,E2 -20653.122} C_VEL
LIN {X 0,Y 215.332,Z 270.414,A -85,B 0,C 180,E1 -20656.733,E2 -20656.733} C_VEL
LIN {X 0,Y 214.536,Z 266.089,A -85,B 0,C 180,E1 -20661.837,E2 -20661.837} C_VEL
LIN {X 0,Y 213.977,Z 262.811,A -85,B 0,C 180,E1 -20666.058,E2 -20666.058} C_VEL
LIN {X 0,Y 213.753,Z 261.858,A -85,B 0,C 180,E1 -20667.705,E2 -20667.705} C_VEL
LIN {X 0,Y 213.797,Z 261.852,A -85,B 0,C 180,E1 -20672.599,E2 -20672.599} C_VEL
LIN {X 0,Y 213.82,Z 261.85,A -85,B 0,C 180,E1 -20676.98,E2 -20676.98} C_VEL
LIN {X 0,Y 213.899,Z 261.841,A -85,B 0,C 180,E1 -20682.8,E2 -20682.8} C_VEL
LIN {X 0,Y 213.923,Z 261.839,A -85,B 0,C 180,E1 -20686.705,E2 -20686.705} C_VEL
LIN {X 0,Y 214.135,Z 261.812,A -85,B 0,C 180,E1 -20690.555,E2 -20690.555} C_VEL
LIN {X 0,Y 214.104,Z 261.816,A -85,B 0,C 180,E1 -20694.349,E2 -20694.349} C_VEL
LIN {X 0,Y 214.453,Z 261.772,A -85,B 0,C 180,E1 -20698.122,E2 -20698.122} C_VEL
LIN {X 0,Y 214.549,Z 261.755,A -85,B 0,C 180,E1 -20700,E2 -20700} C_VEL
LIN {X 0,Y 214.417,Z 261.777,A -85,B 0,C 180,E1 -20701.879,E2 -20701.879} C_VEL
LIN {X 0,Y 214.189,Z 261.805,A -85,B 0,C 180,E1 -20707.542,E2 -20707.542} C_VEL
LIN {X 0,Y 214.003,Z 261.828,A -85,B 0,C 180,E1 -20711.364,E2 -20711.364} C_VEL
LIN {X 0,Y 213.911,Z 261.836,A -85,B 0,C 180,E1 -20715.239,E2 -20715.239} C_VEL
LIN {X 0,Y 213.822,Z 261.846,A -85,B 0,C 180,E1 -20719.189,E2 -20719.189} C_VEL
LIN {X 0,Y 213.773,Z 261.854,A -85,B 0,C 180,E1 -20723.236,E2 -20723.236} C_VEL
LIN {X 0,Y 213.794,Z 261.853,A -85,B 0,C 180,E1 -20727.426,E2 -20727.426} C_VEL
LIN {X 0,Y 213.767,Z 261.856,A -85,B 0,C 180,E1 -20731.738,E2 -20731.738} C_VEL
LIN {X 0,Y 213.752,Z 261.858,A -85,B 0,C 180,E1 -20736.287,E2 -20736.287} C_VEL
LIN {X 0,Y 213.719,Z 261.863,A -85,B 0,C 180,E1 -20741.124,E2 -20741.124} C_VEL
LIN {X 0,Y 213.711,Z 261.863,A -85,B 0,C 180,E1 -20743.678,E2 -20743.678} C_VEL
LIN {X 0,Y 213.709,Z 261.866,A -85,B 0,C 180,E1 -20746.344,E2 -20746.344} C_VEL
LIN {X 0,Y 213.708,Z 261.865,A -85,B 0,C 180,E1 -20751.327,E2 -20751.327} C_VEL
LIN {X 0,Y 213.741,Z 261.861,A -85,B 0,C 180,E1 -20755.289,E2 -20755.289} C_VEL
LIN {X 0,Y 213.566,Z 261.876,A -85,B 0,C 180,E1 -20758.226,E2 -20758.226} C_VEL
LIN {X 0,Y 213.52,Z 263.472,A -85,B 0,C 180,E1 -20760.997,E2 -20760.997} C_VEL
LIN {X 0,Y 214.612,Z 266.553,A -85,B 0,C 180,E1 -20761.368,E2 -20761.368} C_VEL
LIN {X 0,Y 219.073,Z 277.698,A -85,B 0,C 180,E1 -20762.913,E2 -20762.913} C_VEL
LIN {X 0,Y 222.464,Z 289.113,A -85,B 0,C 180,E1 -20764.603,E2 -20764.603} C_VEL
LIN {X 0,Y 224.6,Z 299.056,A -85,B 0,C 180,E1 -20766.229,E2 -20766.229} C_VEL
LIN {X 0,Y 225.746,Z 307.19,A -85,B 0,C 180,E1 -20767.694,E2 -20767.694} C_VEL
LIN {X 0,Y 223.884,Z 317.932,A -85,B 0,C 180,E1 -20769.557,E2 -20769.557} C_VEL
LIN {X 0,Y 221.774,Z 327.173,A -85,B 0,C 180,E1 -20771.522,E2 -20771.522} C_VEL
LIN {X 0,Y 219.62,Z 335.631,A -85,B 0,C 180,E1 -20773.746,E2 -20773.746} C_VEL
LIN {X 0,Y 217.48,Z 343.797,A -85,B 0,C 180,E1 -20776.448,E2 -20776.448} C_VEL
LIN {X 0,Y 215.842,Z 349.418,A -85,B 0,C 180,E1 -20778.731,E2 -20778.731} C_VEL
LIN {X 0,Y 214.869,Z 353.2,A -85,B 0,C 180,E1 -20780.585,E2 -20780.585} C_VEL
LIN {X 0,Y 213.708,Z 357.873,A -85,B 0,C 180,E1 -20783.388,E2 -20783.388} C_VEL
LIN {X 0,Y 212.677,Z 361.47,A -85,B 0,C 180,E1 -20786.208,E2 -20786.208} C_VEL
LIN {X 0,Y 212.287,Z 363.326,A -85,B 0,C 180,E1 -20788.1,E2 -20788.1} C_VEL
LIN {X 0,Y 212.033,Z 364.726,A -85,B 0,C 180,E1 -20789.997,E2 -20789.997} C_VEL
LIN {X 0,Y 211.99,Z 366.34,A -85,B 0,C 180,E1 -20793.799,E2 -20793.799} C_VEL
LIN {X 0,Y 212.133,Z 366.553,A -85,B 0,C 180,E1 -20796.324,E2 -20796.324} C_VEL
LIN {X 0,Y 212.455,Z 365.848,A -85,B 0,C 180,E1 -20799.518,E2 -20799.518} C_VEL
LIN {X 0,Y 213.442,Z 363.556,A -85,B 0,C 180,E1 -20803.323,E2 -20803.323} C_VEL
LIN {X 0,Y 214.663,Z 360.701,A -85,B 0,C 180,E1 -20806.155,E2 -20806.155} C_VEL
LIN {X 0,Y 216.238,Z 356.814,A -85,B 0,C 180,E1 -20808.963,E2 -20808.963} C_VEL
LIN {X 0,Y 218.252,Z 351.778,A -85,B 0,C 180,E1 -20811.732,E2 -20811.732} C_VEL
LIN {X 0,Y 220.742,Z 345.402,A -85,B 0,C 180,E1 -20814.447,E2 -20814.447} C_VEL
LIN {X 0,Y 223.574,Z 337.424,A -85,B 0,C 180,E1 -20817.113,E2 -20817.113} C_VEL
LIN {X 0,Y 226.282,Z 328.828,A -85,B 0,C 180,E1 -20819.408,E2 -20819.408} C_VEL
LIN {X 0,Y 229.081,Z 319.272,A -85,B 0,C 180,E1 -20821.433,E2 -20821.433} C_VEL
LIN {X 0,Y 230.255,Z 314.568,A -85,B 0,C 180,E1 -20822.283,E2 -20822.283} C_VEL
LIN {X 0,Y 228.944,Z 304.971,A -85,B 0,C 180,E1 -20824.333,E2 -20824.333} C_VEL
LIN {X 0,Y 226.696,Z 295.129,A -85,B 0,C 180,E1 -20826.288,E2 -20826.288} C_VEL
LIN {X 0,Y 223.517,Z 285.067,A -85,B 0,C 180,E1 -20828.18,E2 -20828.18} C_VEL
LIN {X 0,Y 219.003,Z 274.388,A -85,B 0,C 180,E1 -20830.157,E2 -20830.157} C_VEL
LIN {X 0,Y 215.75,Z 268.178,A -85,B 0,C 180,E1 -20831.331,E2 -20831.331} C_VEL
LIN {X 0,Y 214.303,Z 265.452,A -85,B 0,C 180,E1 -20831.836,E2 -20831.836} C_VEL
LIN {X 0,Y 214.049,Z 264.384,A -85,B 0,C 180,E1 -20832.025,E2 -20832.025} C_VEL
LIN {X 0,Y 213.77,Z 262.324,A -85,B 0,C 180,E1 -20836.337,E2 -20836.337} C_VEL
LIN {X 0,Y 213.712,Z 261.863,A -85,B 0,C 180,E1 -20839.14,E2 -20839.14} C_VEL
LIN {X 0,Y 213.745,Z 261.857,A -85,B 0,C 180,E1 -20843.711,E2 -20843.711} C_VEL
LIN {X 0,Y 213.788,Z 261.85,A -85,B 0,C 180,E1 -20848.723,E2 -20848.723} C_VEL
LIN {X 0,Y 213.817,Z 261.844,A -85,B 0,C 180,E1 -20852.602,E2 -20852.602} C_VEL
LIN {X 0,Y 213.843,Z 261.848,A -85,B 0,C 180,E1 -20856.951,E2 -20856.951} C_VEL
LIN {X 0,Y 213.934,Z 261.838,A -85,B 0,C 180,E1 -20862.802,E2 -20862.802} C_VEL
LIN {X 0,Y 213.97,Z 261.831,A -85,B 0,C 180,E1 -20866.707,E2 -20866.707} C_VEL
LIN {X 0,Y 214.186,Z 261.804,A -85,B 0,C 180,E1 -20870.557,E2 -20870.557} C_VEL
LIN {X 0,Y 214.239,Z 261.799,A -85,B 0,C 180,E1 -20872.46,E2 -20872.46} C_VEL
LIN {X 0,Y 214.469,Z 261.769,A -85,B 0,C 180,E1 -20878.122,E2 -20878.122} C_VEL
LIN {X 0,Y 214.436,Z 261.774,A -85,B 0,C 180,E1 -20881.878,E2 -20881.878} C_VEL
LIN {X 0,Y 214.238,Z 261.8,A -85,B 0,C 180,E1 -20887.54,E2 -20887.54} C_VEL
LIN {X 0,Y 214.037,Z 261.823,A -85,B 0,C 180,E1 -20891.362,E2 -20891.362} C_VEL
LIN {X 0,Y 213.923,Z 261.829,A -85,B 0,C 180,E1 -20895.238,E2 -20895.238} C_VEL
LIN {X 0,Y 213.829,Z 261.842,A -85,B 0,C 180,E1 -20899.188,E2 -20899.188} C_VEL
LIN {X 0,Y 213.827,Z 261.849,A -85,B 0,C 180,E1 -20904.258,E2 -20904.258} C_VEL
LIN {X 0,Y 213.794,Z 261.869,A -85,B 0,C 180,E1 -20905.299,E2 -20905.299} C_VEL
LIN {X 0,Y 214.25,Z 264.285,A -85,B 0,C 180,E1 -20909.475,E2 -20909.475} C_VEL
LIN {X 0,Y 214.703,Z 267.14,A -85,B 0,C 180,E1 -20913.812,E2 -20913.812} C_VEL
LIN {X 0,Y 215.248,Z 270.489,A -85,B 0,C 180,E1 -20918.412,E2 -20918.412} C_VEL
LIN {X 0,Y 215.955,Z 274.306,A -85,B 0,C 180,E1 -20923.112,E2 -20923.112} C_VEL
LIN {X 0,Y 216.619,Z 277.746,A -85,B 0,C 180,E1 -20927.057,E2 -20927.057} C_VEL
LIN {X 0,Y 217.061,Z 280.146,A -85,B 0,C 180,E1 -20929.646,E2 -20929.646} C_VEL
LIN {X 0,Y 217,Z 283.404,A -85,B 0,C 180,E1 -20932.939,E2 -20932.939} C_VEL
LIN {X 0,Y 218.154,Z 287.281,A -85,B 0,C 180,E1 -20933.445,E2 -20933.445} C_VEL
LIN {X 0,Y 221.531,Z 299.271,A -85,B 0,C 180,E1 -20935.034,E2 -20935.034} C_VEL
LIN {X 0,Y 223.987,Z 311.33,A -85,B 0,C 180,E1 -20936.766,E2 -20936.766} C_VEL
LIN {X 0,Y 225.287,Z 322.689,A -85,B 0,C 180,E1 -20938.544,E2 -20938.544} C_VEL
LIN {X 0,Y 225.778,Z 333.17,A -85,B 0,C 180,E1 -20940.395,E2 -20940.395} C_VEL
LIN {X 0,Y 225.562,Z 341.232,A -85,B 0,C 180,E1 -20941.989,E2 -20941.989} C_VEL
LIN {X 0,Y 224.979,Z 344.31,A -85,B 0,C 180,E1 -20942.593,E2 -20942.593} C_VEL
LIN {X 0,Y 223.745,Z 347.353,A -85,B 0,C 180,E1 -20943.151,E2 -20943.151} C_VEL
LIN {X 0,Y 220.135,Z 353.137,A -85,B 0,C 180,E1 -20944.21,E2 -20944.21} C_VEL
LIN {X 0,Y 215.253,Z 359.928,A -85,B 0,C 180,E1 -20945.694,E2 -20945.694} C_VEL
LIN {X 0,Y 213.269,Z 363.737,A -85,B 0,C 180,E1 -20946.814,E2 -20946.814} C_VEL
LIN {X 0,Y 210.763,Z 371.112,A -85,B 0,C 180,E1 -20949.519,E2 -20949.519} C_VEL
LIN {X 0,Y 208.532,Z 377.246,A -85,B 0,C 180,E1 -20952.346,E2 -20952.346} C_VEL
LIN {X 0,Y 206.745,Z 382.148,A -85,B 0,C 180,E1 -20955.232,E2 -20955.232} C_VEL
LIN {X 0,Y 205.571,Z 385.945,A -85,B 0,C 180,E1 -20958.166,E2 -20958.166} C_VEL
LIN {X 0,Y 205.077,Z 387.92,A -85,B 0,C 180,E1 -20960.137,E2 -20960.137} C_VEL
LIN {X 0,Y 204.735,Z 389.475,A -85,B 0,C 180,E1 -20962.111,E2 -20962.111} C_VEL
LIN {X 0,Y 204.576,Z 390.992,A -85,B 0,C 180,E1 -20965.046,E2 -20965.046} C_VEL
LIN {X 0,Y 204.653,Z 391.619,A -85,B 0,C 180,E1 -20968.035,E2 -20968.035} C_VEL
LIN {X 0,Y 204.739,Z 391.545,A -85,B 0,C 180,E1 -20970.003,E2 -20970.003} C_VEL
LIN {X 0,Y 204.7,Z 391.019,A -85,B 0,C 180,E1 -20971.97,E2 -20971.97} C_VEL
LIN {X 0,Y 204.603,Z 389.395,A -85,B 0,C 180,E1 -20975.039,E2 -20975.039} C_VEL
LIN {X 0,Y 204.929,Z 385.895,A -85,B 0,C 180,E1 -20978.881,E2 -20978.881} C_VEL
LIN {X 0,Y 205.567,Z 382.01,A -85,B 0,C 180,E1 -20981.84,E2 -20981.84} C_VEL
LIN {X 0,Y 206.706,Z 376.993,A -85,B 0,C 180,E1 -20984.776,E2 -20984.776} C_VEL
LIN {X 0,Y 208.303,Z 370.686,A -85,B 0,C 180,E1 -20987.68,E2 -20987.68} C_VEL
LIN {X 0,Y 209.977,Z 364.495,A -85,B 0,C 180,E1 -20989.973,E2 -20989.973} C_VEL
LIN {X 0,Y 212.034,Z 356.51,A -85,B 0,C 180,E1 -20992.409,E2 -20992.409} C_VEL
LIN {X 0,Y 214.435,Z 347.121,A -85,B 0,C 180,E1 -20994.703,E2 -20994.703} C_VEL
LIN {X 0,Y 214.994,Z 342.71,A -85,B 0,C 180,E1 -20995.669,E2 -20995.669} C_VEL
LIN {X 0,Y 215.289,Z 332.277,A -85,B 0,C 180,E1 -20997.734,E2 -20997.734} C_VEL
LIN {X 0,Y 214.959,Z 320.858,A -85,B 0,C 180,E1 -20999.647,E2 -20999.647} C_VEL
LIN {X 0,Y 213.897,Z 309.123,A -85,B 0,C 180,E1 -21001.32,E2 -21001.32} C_VEL
LIN {X 0,Y 211.906,Z 297.166,A -85,B 0,C 180,E1 -21002.801,E2 -21002.801} C_VEL
LIN {X 0,Y 208.806,Z 284.699,A -85,B 0,C 180,E1 -21004.155,E2 -21004.155} C_VEL
LIN {X 0,Y 208.718,Z 283.632,A -85,B 0,C 180,E1 -21004.266,E2 -21004.266} C_VEL
LIN {X 0,Y 209.528,Z 280.587,A -85,B 0,C 180,E1 -21007.143,E2 -21007.143} C_VEL
LIN {X 0,Y 209.492,Z 278.174,A -85,B 0,C 180,E1 -21009.602,E2 -21009.602} C_VEL
LIN {X 0,Y 208.838,Z 274.379,A -85,B 0,C 180,E1 -21013.653,E2 -21013.653} C_VEL
LIN {X 0,Y 208.118,Z 270.548,A -85,B 0,C 180,E1 -21017.985,E2 -21017.985} C_VEL
LIN {X 0,Y 207.473,Z 266.995,A -85,B 0,C 180,E1 -21022.43,E2 -21022.43} C_VEL
LIN {X 0,Y 207.199,Z 265.206,A -85,B 0,C 180,E1 -21024.787,E2 -21024.787} C_VEL
LIN {X 0,Y 206.73,Z 262.733,A -85,B 0,C 180,E1 -21028.384,E2 -21028.384} C_VEL
LIN {X 0,Y 206.714,Z 262.735,A -85,B 0,C 180,E1 -21033.77,E2 -21033.77} C_VEL
LIN {X 0,Y 206.74,Z 262.733,A -85,B 0,C 180,E1 -21038.041,E2 -21038.041} C_VEL
LIN {X 0,Y 206.833,Z 262.723,A -85,B 0,C 180,E1 -21042.193,E2 -21042.193} C_VEL
LIN {X 0,Y 206.864,Z 262.72,A -85,B 0,C 180,E1 -21046.242,E2 -21046.242} C_VEL
LIN {X 0,Y 207.081,Z 262.692,A -85,B 0,C 180,E1 -21050.23,E2 -21050.23} C_VEL
LIN {X 0,Y 207.065,Z 262.693,A -85,B 0,C 180,E1 -21054.156,E2 -21054.156} C_VEL
LIN {X 0,Y 207.389,Z 262.652,A -85,B 0,C 180,E1 -21058.058,E2 -21058.058} C_VEL
LIN {X 0,Y 207.514,Z 262.631,A -85,B 0,C 180,E1 -21060,E2 -21060} C_VEL
LIN {X 0,Y 207.056,Z 262.69,A -85,B 0,C 180,E1 -21063.893,E2 -21063.893} C_VEL
LIN {X 0,Y 207.134,Z 262.682,A -85,B 0,C 180,E1 -21067.8,E2 -21067.8} C_VEL
LIN {X 0,Y 206.925,Z 262.709,A -85,B 0,C 180,E1 -21071.759,E2 -21071.759} C_VEL
LIN {X 0,Y 206.839,Z 262.718,A -85,B 0,C 180,E1 -21075.773,E2 -21075.773} C_VEL
LIN {X 0,Y 206.74,Z 262.726,A -85,B 0,C 180,E1 -21079.874,E2 -21079.874} C_VEL
LIN {X 0,Y 206.7,Z 262.734,A -85,B 0,C 180,E1 -21084.08,E2 -21084.08} C_VEL
LIN {X 0,Y 206.695,Z 262.736,A -85,B 0,C 180,E1 -21088.427,E2 -21088.427} C_VEL
LIN {X 0,Y 206.704,Z 262.734,A -85,B 0,C 180,E1 -21092.957,E2 -21092.957} C_VEL
LIN {X 0,Y 206.688,Z 262.737,A -85,B 0,C 180,E1 -21097.739,E2 -21097.739} C_VEL
LIN {X 0,Y 206.649,Z 262.744,A -85,B 0,C 180,E1 -21101.561,E2 -21101.561} C_VEL
LIN {X 0,Y 206.638,Z 262.744,A -85,B 0,C 180,E1 -21105.581,E2 -21105.581} C_VEL
LIN {X 0,Y 206.653,Z 262.744,A -85,B 0,C 180,E1 -21109.744,E2 -21109.744} C_VEL
LIN {X 0,Y 206.689,Z 262.739,A -85,B 0,C 180,E1 -21114.694,E2 -21114.694} C_VEL
LIN {X 0,Y 206.57,Z 262.75,A -85,B 0,C 180,E1 -21117.016,E2 -21117.016} C_VEL
LIN {X 0,Y 206.533,Z 263.647,A -85,B 0,C 180,E1 -21119.305,E2 -21119.305} C_VEL
LIN {X 0,Y 206.532,Z 263.917,A -85,B 0,C 180,E1 -21119.785,E2 -21119.785} C_VEL
LIN {X 0,Y 207.764,Z 267.205,A -85,B 0,C 180,E1 -21120.239,E2 -21120.239} C_VEL
LIN {X 0,Y 212.595,Z 279.04,A -85,B 0,C 180,E1 -21122.004,E2 -21122.004} C_VEL
LIN {X 0,Y 215.985,Z 290.529,A -85,B 0,C 180,E1 -21123.812,E2 -21123.812} C_VEL
LIN {X 0,Y 218.284,Z 301.842,A -85,B 0,C 180,E1 -21125.786,E2 -21125.786} C_VEL
LIN {X 0,Y 219.184,Z 309.169,A -85,B 0,C 180,E1 -21127.184,E2 -21127.184} C_VEL
LIN {X 0,Y 217.073,Z 319.85,A -85,B 0,C 180,E1 -21129.134,E2 -21129.134} C_VEL
LIN {X 0,Y 214.584,Z 329.687,A -85,B 0,C 180,E1 -21131.375,E2 -21131.375} C_VEL
LIN {X 0,Y 212.196,Z 338.737,A -85,B 0,C 180,E1 -21133.981,E2 -21133.981} C_VEL
LIN {X 0,Y 210.035,Z 346.779,A -85,B 0,C 180,E1 -21136.944,E2 -21136.944} C_VEL
LIN {X 0,Y 208.921,Z 350.009,A -85,B 0,C 180,E1 -21138.353,E2 -21138.353} C_VEL
LIN {X 0,Y 208.571,Z 351.97,A -85,B 0,C 180,E1 -21139.317,E2 -21139.317} C_VEL
LIN {X 0,Y 206.903,Z 357.02,A -85,B 0,C 180,E1 -21142.188,E2 -21142.188} C_VEL
LIN {X 0,Y 205.945,Z 360.925,A -85,B 0,C 180,E1 -21145.103,E2 -21145.103} C_VEL
LIN {X 0,Y 205.208,Z 363.821,A -85,B 0,C 180,E1 -21148.034,E2 -21148.034} C_VEL
LIN {X 0,Y 204.875,Z 366.181,A -85,B 0,C 180,E1 -21151.963,E2 -21151.963} C_VEL
LIN {X 0,Y 204.91,Z 366.787,A -85,B 0,C 180,E1 -21153.93,E2 -21153.93} C_VEL
LIN {X 0,Y 205.069,Z 366.987,A -85,B 0,C 180,E1 -21156.342,E2 -21156.342} C_VEL
LIN {X 0,Y 205.428,Z 366.243,A -85,B 0,C 180,E1 -21159.846,E2 -21159.846} C_VEL
LIN {X 0,Y 205.882,Z 365.281,A -85,B 0,C 180,E1 -21161.816,E2 -21161.816} C_VEL
LIN {X 0,Y 206.499,Z 363.919,A -85,B 0,C 180,E1 -21163.78,E2 -21163.78} C_VEL
LIN {X 0,Y 207.822,Z 361.04,A -85,B 0,C 180,E1 -21166.702,E2 -21166.702} C_VEL
LIN {X 0,Y 209.497,Z 357.124,A -85,B 0,C 180,E1 -21169.598,E2 -21169.598} C_VEL
LIN {X 0,Y 211.63,Z 352.05,A -85,B 0,C 180,E1 -21172.448,E2 -21172.448} C_VEL
LIN {X 0,Y 214.26,Z 345.627,A -85,B 0,C 180,E1 -21175.237,E2 -21175.237} C_VEL
LIN {X 0,Y 217.257,Z 337.606,A -85,B 0,C 180,E1 -21177.97,E2 -21177.97} C_VEL
LIN {X 0,Y 219.918,Z 329.501,A -85,B 0,C 180,E1 -21180.186,E2 -21180.186} C_VEL
LIN {X 0,Y 223.043,Z 319.322,A -85,B 0,C 180,E1 -21182.386,E2 -21182.386} C_VEL
LIN {X 0,Y 223.804,Z 316.084,A -85,B 0,C 180,E1 -21182.999,E2 -21182.999} C_VEL
LIN {X 0,Y 222.534,Z 306.189,A -85,B 0,C 180,E1 -21185.232,E2 -21185.232} C_VEL
LIN {X 0,Y 220.301,Z 296.331,A -85,B 0,C 180,E1 -21187.307,E2 -21187.307} C_VEL
LIN {X 0,Y 217.445,Z 287.249,A -85,B 0,C 180,E1 -21189.131,E2 -21189.131} C_VEL
LIN {X 0,Y 213.187,Z 276.966,A -85,B 0,C 180,E1 -21191.182,E2 -21191.182} C_VEL
LIN {X 0,Y 208.843,Z 268.881,A -85,B 0,C 180,E1 -21192.872,E2 -21192.872} C_VEL
LIN {X 0,Y 207.232,Z 265.988,A -85,B 0,C 180,E1 -21193.47,E2 -21193.47} C_VEL
LIN {X 0,Y 206.961,Z 264.935,A -85,B 0,C 180,E1 -21193.636,E2 -21193.636} C_VEL
LIN {X 0,Y 206.653,Z 262.812,A -85,B 0,C 180,E1 -21198.429,E2 -21198.429} C_VEL
LIN {X 0,Y 206.692,Z 262.74,A -85,B 0,C 180,E1 -21202.262,E2 -21202.262} C_VEL
LIN {X 0,Y 206.724,Z 262.736,A -85,B 0,C 180,E1 -21204.693,E2 -21204.693} C_VEL
LIN {X 0,Y 206.715,Z 262.73,A -85,B 0,C 180,E1 -21209.337,E2 -21209.337} C_VEL
LIN {X 0,Y 206.724,Z 262.733,A -85,B 0,C 180,E1 -21213.771,E2 -21213.771} C_VEL
LIN {X 0,Y 206.749,Z 262.732,A -85,B 0,C 180,E1 -21218.042,E2 -21218.042} C_VEL
LIN {X 0,Y 206.864,Z 262.716,A -85,B 0,C 180,E1 -21222.195,E2 -21222.195} C_VEL
LIN {X 0,Y 206.904,Z 262.71,A -85,B 0,C 180,E1 -21226.245,E2 -21226.245} C_VEL
LIN {X 0,Y 207.123,Z 262.685,A -85,B 0,C 180,E1 -21230.232,E2 -21230.232} C_VEL
LIN {X 0,Y 207.179,Z 262.68,A -85,B 0,C 180,E1 -21232.201,E2 -21232.201} C_VEL
LIN {X 0,Y 207.402,Z 262.649,A -85,B 0,C 180,E1 -21238.058,E2 -21238.058} C_VEL
LIN {X 0,Y 207.501,Z 262.637,A -85,B 0,C 180,E1 -21240,E2 -21240} C_VEL
LIN {X 0,Y 207.373,Z 262.654,A -85,B 0,C 180,E1 -21241.942,E2 -21241.942} C_VEL
LIN {X 0,Y 207.179,Z 262.679,A -85,B 0,C 180,E1 -21247.798,E2 -21247.798} C_VEL
LIN {X 0,Y 206.973,Z 262.704,A -85,B 0,C 180,E1 -21251.755,E2 -21251.755} C_VEL
LIN {X 0,Y 206.856,Z 262.709,A -85,B 0,C 180,E1 -21255.771,E2 -21255.771} C_VEL
LIN {X 0,Y 206.774,Z 262.723,A -85,B 0,C 180,E1 -21259.87,E2 -21259.87} C_VEL
LIN {X 0,Y 206.803,Z 262.903,A -85,B 0,C 180,E1 -21264.067,E2 -21264.067} C_VEL
LIN {X 0,Y 207.187,Z 265.24,A -85,B 0,C 180,E1 -21268.352,E2 -21268.352} C_VEL
LIN {X 0,Y 207.653,Z 267.968,A -85,B 0,C 180,E1 -21272.787,E2 -21272.787} C_VEL
LIN {X 0,Y 208.158,Z 271.222,A -85,B 0,C 180,E1 -21277.425,E2 -21277.425} C_VEL
LIN {X 0,Y 208.834,Z 274.946,A -85,B 0,C 180,E1 -21282.305,E2 -21282.305} C_VEL
LIN {X 0,Y 209.489,Z 278.212,A -85,B 0,C 180,E1 -21286.228,E2 -21286.228} C_VEL
LIN {X 0,Y 210.094,Z 281.849,A -85,B 0,C 180,E1 -21290.299,E2 -21290.299} C_VEL
LIN {X 0,Y 210.133,Z 283.168,A -85,B 0,C 180,E1 -21291.463,E2 -21291.463} C_VEL
LIN {X 0,Y 211.279,Z 286.635,A -85,B 0,C 180,E1 -21291.936,E2 -21291.936} C_VEL
LIN {X 0,Y 212.24,Z 288.977,A -85,B 0,C 180,E1 -21292.306,E2 -21292.306} C_VEL
LIN {X 0,Y 215.213,Z 299.496,A -85,B 0,C 180,E1 -21293.826,E2 -21293.826} C_VEL
LIN {X 0,Y 217.652,Z 311.44,A -85,B 0,C 180,E1 -21295.654,E2 -21295.654} C_VEL
LIN {X 0,Y 218.926,Z 322.753,A -85,B 0,C 180,E1 -21297.52,E2 -21297.52} C_VEL
LIN {X 0,Y 219.336,Z 333.656,A -85,B 0,C 180,E1 -21299.539,E2 -21299.539} C_VEL
LIN {X 0,Y 218.846,Z 344.063,A -85,B 0,C 180,E1 -21301.73,E2 -21301.73} C_VEL
LIN {X 0,Y 218.34,Z 348.268,A -85,B 0,C 180,E1 -21302.701,E2 -21302.701} C_VEL
LIN {X 0,Y 215.427,Z 357.324,A -85,B 0,C 180,E1 -21304.909,E2 -21304.909} C_VEL
LIN {X 0,Y 213.269,Z 363.737,A -85,B 0,C 180,E1 -21306.814,E2 -21306.814} C_VEL
LIN {X 0,Y 211.393,Z 367.339,A -85,B 0,C 180,E1 -21307.994,E2 -21307.994} C_VEL
LIN {X 0,Y 206.743,Z 372.705,A -85,B 0,C 180,E1 -21309.903,E2 -21309.903} C_VEL
LIN {X 0,Y 202.231,Z 377.361,A -85,B 0,C 180,E1 -21311.995,E2 -21311.995} C_VEL
LIN {X 0,Y 200.609,Z 379.883,A -85,B 0,C 180,E1 -21313.433,E2 -21313.433} C_VEL
LIN {X 0,Y 198.941,Z 384.465,A -85,B 0,C 180,E1 -21316.728,E2 -21316.728} C_VEL
LIN {X 0,Y 198.039,Z 387.55,A -85,B 0,C 180,E1 -21319.782,E2 -21319.782} C_VEL
LIN {X 0,Y 197.683,Z 389.087,A -85,B 0,C 180,E1 -21321.827,E2 -21321.827} C_VEL
LIN {X 0,Y 197.497,Z 390.681,A -85,B 0,C 180,E1 -21325.13,E2 -21325.13} C_VEL
LIN {X 0,Y 197.562,Z 391.197,A -85,B 0,C 180,E1 -21327.964,E2 -21327.964} C_VEL
LIN {X 0,Y 197.671,Z 391.108,A -85,B 0,C 180,E1 -21330.003,E2 -21330.003} C_VEL
LIN {X 0,Y 197.608,Z 390.564,A -85,B 0,C 180,E1 -21332.041,E2 -21332.041} C_VEL
LIN {X 0,Y 197.529,Z 389.093,A -85,B 0,C 180,E1 -21334.979,E2 -21334.979} C_VEL
LIN {X 0,Y 197.902,Z 385.393,A -85,B 0,C 180,E1 -21339.199,E2 -21339.199} C_VEL
LIN {X 0,Y 198.583,Z 381.482,A -85,B 0,C 180,E1 -21342.263,E2 -21342.263} C_VEL
LIN {X 0,Y 199.81,Z 376.438,A -85,B 0,C 180,E1 -21345.299,E2 -21345.299} C_VEL
LIN {X 0,Y 201.502,Z 370.101,A -85,B 0,C 180,E1 -21348.298,E2 -21348.298} C_VEL
LIN {X 0,Y 202.988,Z 365.001,A -85,B 0,C 180,E1 -21350.26,E2 -21350.26} C_VEL
LIN {X 0,Y 204.991,Z 357.501,A -85,B 0,C 180,E1 -21352.69,E2 -21352.69} C_VEL
LIN {X 0,Y 207.695,Z 347.443,A -85,B 0,C 180,E1 -21355.293,E2 -21355.293} C_VEL
LIN {X 0,Y 208.291,Z 341.919,A -85,B 0,C 180,E1 -21356.559,E2 -21356.559} C_VEL
LIN {X 0,Y 208.673,Z 330.428,A -85,B 0,C 180,E1 -21358.876,E2 -21358.876} C_VEL
LIN {X 0,Y 208.262,Z 318.737,A -85,B 0,C 180,E1 -21360.874,E2 -21360.874} C_VEL
LIN {X 0,Y 207.035,Z 306.75,A -85,B 0,C 180,E1 -21362.618,E2 -21362.618} C_VEL
LIN {X 0,Y 204.732,Z 294.423,A -85,B 0,C 180,E1 -21364.19,E2 -21364.19} C_VEL
LIN {X 0,Y 201.98,Z 283.182,A -85,B 0,C 180,E1 -21365.451,E2 -21365.451} C_VEL
LIN {X 0,Y 202.41,Z 281.628,A -85,B 0,C 180,E1 -21367.004,E2 -21367.004} C_VEL
LIN {X 0,Y 202.542,Z 280.035,A -85,B 0,C 180,E1 -21368.655,E2 -21368.655} C_VEL
LIN {X 0,Y 201.91,Z 276.057,A -85,B 0,C 180,E1 -21373.033,E2 -21373.033} C_VEL
LIN {X 0,Y 201.255,Z 272.47,A -85,B 0,C 180,E1 -21377.171,E2 -21377.171} C_VEL
LIN {X 0,Y 200.718,Z 269.501,A -85,B 0,C 180,E1 -21380.931,E2 -21380.931} C_VEL
LIN {X 0,Y 200.076,Z 265.914,A -85,B 0,C 180,E1 -21385.804,E2 -21385.804} C_VEL
LIN {X 0,Y 199.666,Z 263.612,A -85,B 0,C 180,E1 -21389.311,E2 -21389.311} C_VEL
LIN {X 0,Y 199.652,Z 263.614,A -85,B 0,C 180,E1 -21392.767,E2 -21392.767} C_VEL
LIN {X 0,Y 199.716,Z 263.607,A -85,B 0,C 180,E1 -21397.227,E2 -21397.227} C_VEL
LIN {X 0,Y 199.758,Z 263.603,A -85,B 0,C 180,E1 -21401.8,E2 -21401.8} C_VEL
LIN {X 0,Y 199.804,Z 263.599,A -85,B 0,C 180,E1 -21405.746,E2 -21405.746} C_VEL
LIN {X 0,Y 200.032,Z 263.571,A -85,B 0,C 180,E1 -21409.882,E2 -21409.882} C_VEL
LIN {X 0,Y 200.027,Z 263.571,A -85,B 0,C 180,E1 -21413.95,E2 -21413.95} C_VEL
LIN {X 0,Y 200.329,Z 263.532,A -85,B 0,C 180,E1 -21417.99,E2 -21417.99} C_VEL
LIN {X 0,Y 200.478,Z 263.508,A -85,B 0,C 180,E1 -21420,E2 -21420} C_VEL
LIN {X 0,Y 200.002,Z 263.568,A -85,B 0,C 180,E1 -21424.03,E2 -21424.03} C_VEL
LIN {X 0,Y 200.082,Z 263.56,A -85,B 0,C 180,E1 -21428.077,E2 -21428.077} C_VEL
LIN {X 0,Y 199.875,Z 263.587,A -85,B 0,C 180,E1 -21432.18,E2 -21432.18} C_VEL
LIN {X 0,Y 199.776,Z 263.598,A -85,B 0,C 180,E1 -21436.346,E2 -21436.346} C_VEL
LIN {X 0,Y 199.665,Z 263.609,A -85,B 0,C 180,E1 -21440.609,E2 -21440.609} C_VEL
LIN {X 0,Y 199.63,Z 263.614,A -85,B 0,C 180,E1 -21444.991,E2 -21444.991} C_VEL
LIN {X 0,Y 199.616,Z 263.616,A -85,B 0,C 180,E1 -21449.532,E2 -21449.532} C_VEL
LIN {X 0,Y 199.674,Z 263.612,A -85,B 0,C 180,E1 -21452.351,E2 -21452.351} C_VEL
LIN {X 0,Y 199.632,Z 263.616,A -85,B 0,C 180,E1 -21456.762,E2 -21456.762} C_VEL
LIN {X 0,Y 199.616,Z 263.618,A -85,B 0,C 180,E1 -21459.327,E2 -21459.327} C_VEL
LIN {X 0,Y 199.581,Z 263.624,A -85,B 0,C 180,E1 -21462.308,E2 -21462.308} C_VEL
LIN {X 0,Y 199.584,Z 263.622,A -85,B 0,C 180,E1 -21465.226,E2 -21465.226} C_VEL
LIN {X 0,Y 199.577,Z 263.624,A -85,B 0,C 180,E1 -21468.001,E2 -21468.001} C_VEL
LIN {X 0,Y 199.603,Z 263.622,A -85,B 0,C 180,E1 -21470.771,E2 -21470.771} C_VEL
LIN {X 0,Y 199.605,Z 263.622,A -85,B 0,C 180,E1 -21474.079,E2 -21474.079} C_VEL
LIN {X 0,Y 199.537,Z 263.968,A -85,B 0,C 180,E1 -21477.707,E2 -21477.707} C_VEL
LIN {X 0,Y 199.584,Z 264.549,A -85,B 0,C 180,E1 -21478.541,E2 -21478.541} C_VEL
LIN {X 0,Y 200.853,Z 267.781,A -85,B 0,C 180,E1 -21478.999,E2 -21478.999} C_VEL
LIN {X 0,Y 205.059,Z 277.615,A -85,B 0,C 180,E1 -21480.577,E2 -21480.577} C_VEL
LIN {X 0,Y 208.362,Z 287.575,A -85,B 0,C 180,E1 -21482.229,E2 -21482.229} C_VEL
LIN {X 0,Y 210.914,Z 298.227,A -85,B 0,C 180,E1 -21484.118,E2 -21484.118} C_VEL
LIN {X 0,Y 212.55,Z 309.159,A -85,B 0,C 180,E1 -21486.255,E2 -21486.255} C_VEL
LIN {X 0,Y 212.001,Z 313.603,A -85,B 0,C 180,E1 -21487.072,E2 -21487.072} C_VEL
LIN {X 0,Y 209.721,Z 323.803,A -85,B 0,C 180,E1 -21489.139,E2 -21489.139} C_VEL
LIN {X 0,Y 207.444,Z 332.165,A -85,B 0,C 180,E1 -21491.222,E2 -21491.222} C_VEL
LIN {X 0,Y 204.871,Z 341.216,A -85,B 0,C 180,E1 -21494.069,E2 -21494.069} C_VEL
LIN {X 0,Y 202.754,Z 348.498,A -85,B 0,C 180,E1 -21496.976,E2 -21496.976} C_VEL
LIN {X 0,Y 201.639,Z 352.547,A -85,B 0,C 180,E1 -21498.945,E2 -21498.945} C_VEL
LIN {X 0,Y 199.896,Z 357.564,A -85,B 0,C 180,E1 -21501.913,E2 -21501.913} C_VEL
LIN {X 0,Y 198.886,Z 361.44,A -85,B 0,C 180,E1 -21504.929,E2 -21504.929} C_VEL
LIN {X 0,Y 198.132,Z 364.312,A -85,B 0,C 180,E1 -21507.964,E2 -21507.964} C_VEL
LIN {X 0,Y 197.806,Z 366.64,A -85,B 0,C 180,E1 -21512.033,E2 -21512.033} C_VEL
LIN {X 0,Y 197.834,Z 367.234,A -85,B 0,C 180,E1 -21514.071,E2 -21514.071} C_VEL
LIN {X 0,Y 197.988,Z 367.426,A -85,B 0,C 180,E1 -21516.317,E2 -21516.317} C_VEL
LIN {X 0,Y 198.424,Z 366.638,A -85,B 0,C 180,E1 -21520.198,E2 -21520.198} C_VEL
LIN {X 0,Y 198.901,Z 365.664,A -85,B 0,C 180,E1 -21522.237,E2 -21522.237} C_VEL
LIN {X 0,Y 199.58,Z 364.278,A -85,B 0,C 180,E1 -21524.267,E2 -21524.267} C_VEL
LIN {X 0,Y 201.005,Z 361.375,A -85,B 0,C 180,E1 -21527.286,E2 -21527.286} C_VEL
LIN {X 0,Y 202.786,Z 357.429,A -85,B 0,C 180,E1 -21530.275,E2 -21530.275} C_VEL
LIN {X 0,Y 205.485,Z 351.315,A -85,B 0,C 180,E1 -21533.692,E2 -21533.692} C_VEL
LIN {X 0,Y 208.306,Z 344.627,A -85,B 0,C 180,E1 -21536.551,E2 -21536.551} C_VEL
LIN {X 0,Y 211.516,Z 336.291,A -85,B 0,C 180,E1 -21539.343,E2 -21539.343} C_VEL
LIN {X 0,Y 214.415,Z 327.667,A -85,B 0,C 180,E1 -21541.627,E2 -21541.627} C_VEL
LIN {X 0,Y 217.059,Z 319.361,A -85,B 0,C 180,E1 -21543.393,E2 -21543.393} C_VEL
LIN {X 0,Y 217.406,Z 317.535,A -85,B 0,C 180,E1 -21543.765,E2 -21543.765} C_VEL
LIN {X 0,Y 216.256,Z 308.078,A -85,B 0,C 180,E1 -21546.026,E2 -21546.026} C_VEL
LIN {X 0,Y 213.948,Z 297.461,A -85,B 0,C 180,E1 -21548.397,E2 -21548.397} C_VEL
LIN {X 0,Y 210.558,Z 287.13,A -85,B 0,C 180,E1 -21550.634,E2 -21550.634} C_VEL
LIN {X 0,Y 206.314,Z 277.533,A -85,B 0,C 180,E1 -21552.734,E2 -21552.734} C_VEL
LIN {X 0,Y 204.082,Z 273.4,A -85,B 0,C 180,E1 -21553.682,E2 -21553.682} C_VEL
LIN {X 0,Y 202.054,Z 269.739,A -85,B 0,C 180,E1 -21554.517,E2 -21554.517} C_VEL
LIN {X 0,Y 200.329,Z 267.112,A -85,B 0,C 180,E1 -21555.176,E2 -21555.176} C_VEL
LIN {X 0,Y 199.867,Z 265.472,A -85,B 0,C 180,E1 -21555.474,E2 -21555.474} C_VEL
LIN {X 0,Y 199.707,Z 264.397,A -85,B 0,C 180,E1 -21558.037,E2 -21558.037} C_VEL
LIN {X 0,Y 199.634,Z 263.616,A -85,B 0,C 180,E1 -21560.754,E2 -21560.754} C_VEL
LIN {X 0,Y 199.626,Z 263.615,A -85,B 0,C 180,E1 -21565.716,E2 -21565.716} C_VEL
LIN {X 0,Y 199.696,Z 263.609,A -85,B 0,C 180,E1 -21568.136,E2 -21568.136} C_VEL
LIN {X 0,Y 199.678,Z 263.605,A -85,B 0,C 180,E1 -21572.77,E2 -21572.77} C_VEL
LIN {X 0,Y 199.729,Z 263.605,A -85,B 0,C 180,E1 -21577.228,E2 -21577.228} C_VEL
LIN {X 0,Y 199.787,Z 263.597,A -85,B 0,C 180,E1 -21581.756,E2 -21581.756} C_VEL
LIN {X 0,Y 199.838,Z 263.591,A -85,B 0,C 180,E1 -21585.748,E2 -21585.748} C_VEL
LIN {X 0,Y 200.066,Z 263.565,A -85,B 0,C 180,E1 -21589.884,E2 -21589.884} C_VEL
LIN {X 0,Y 200.033,Z 263.569,A -85,B 0,C 180,E1 -21593.949,E2 -21593.949} C_VEL
LIN {X 0,Y 200.338,Z 263.529,A -85,B 0,C 180,E1 -21597.989,E2 -21597.989} C_VEL
LIN {X 0,Y 200.466,Z 263.514,A -85,B 0,C 180,E1 -21600,E2 -21600} C_VEL
LIN {X 0,Y 200.025,Z 263.568,A -85,B 0,C 180,E1 -21604.029,E2 -21604.029} C_VEL
LIN {X 0,Y 200.122,Z 263.558,A -85,B 0,C 180,E1 -21608.075,E2 -21608.075} C_VEL
LIN {X 0,Y 199.904,Z 263.583,A -85,B 0,C 180,E1 -21612.177,E2 -21612.177} C_VEL
LIN {X 0,Y 199.794,Z 263.59,A -85,B 0,C 180,E1 -21616.344,E2 -21616.344} C_VEL
LIN {X 0,Y 199.69,Z 263.612,A -85,B 0,C 180,E1 -21620.606,E2 -21620.606} C_VEL
LIN {X 0,Y 199.718,Z 263.711,A -85,B 0,C 180,E1 -21622.227,E2 -21622.227} C_VEL
LIN {X 0,Y 199.946,Z 265.029,A -85,B 0,C 180,E1 -21624.948,E2 -21624.948} C_VEL
LIN {X 0,Y 200.351,Z 267.486,A -85,B 0,C 180,E1 -21629.413,E2 -21629.413} C_VEL
LIN {X 0,Y 200.74,Z 269.538,A -85,B 0,C 180,E1 -21632.839,E2 -21632.839} C_VEL
LIN {X 0,Y 201.102,Z 272.004,A -85,B 0,C 180,E1 -21636.512,E2 -21636.512} C_VEL
LIN {X 0,Y 201.711,Z 275.609,A -85,B 0,C 180,E1 -21641.452,E2 -21641.452} C_VEL
LIN {X 0,Y 202.48,Z 279.27,A -85,B 0,C 180,E1 -21646.042,E2 -21646.042} C_VEL
LIN {X 0,Y 203.013,Z 282.419,A -85,B 0,C 180,E1 -21649.711,E2 -21649.711} C_VEL
LIN {X 0,Y 204.247,Z 285.947,A -85,B 0,C 180,E1 -21650.247,E2 -21650.247} C_VEL
LIN {X 0,Y 205.369,Z 288.166,A -85,B 0,C 180,E1 -21650.677,E2 -21650.677} C_VEL
LIN {X 0,Y 207.766,Z 294.875,A -85,B 0,C 180,E1 -21651.79,E2 -21651.79} C_VEL
LIN {X 0,Y 210.462,Z 306.674,A -85,B 0,C 180,E1 -21653.645,E2 -21653.645} C_VEL
LIN {X 0,Y 212.164,Z 317.858,A -85,B 0,C 180,E1 -21655.542,E2 -21655.542} C_VEL
LIN {X 0,Y 212.804,Z 327.859,A -85,B 0,C 180,E1 -21657.368,E2 -21657.368} C_VEL
LIN {X 0,Y 212.832,Z 337.944,A -85,B 0,C 180,E1 -21659.438,E2 -21659.438} C_VEL
LIN {X 0,Y 212.05,Z 347.123,A -85,B 0,C 180,E1 -21661.551,E2 -21661.551} C_VEL
LIN {X 0,Y 210.865,Z 351.943,A -85,B 0,C 180,E1 -21662.727,E2 -21662.727} C_VEL
LIN {X 0,Y 207.876,Z 360.274,A -85,B 0,C 180,E1 -21665.004,E2 -21665.004} C_VEL
LIN {X 0,Y 204.896,Z 368.454,A -85,B 0,C 180,E1 -21667.836,E2 -21667.836} C_VEL
LIN {X 0,Y 202.432,Z 375.061,A -85,B 0,C 180,E1 -21670.745,E2 -21670.745} C_VEL
LIN {X 0,Y 200.609,Z 379.883,A -85,B 0,C 180,E1 -21673.433,E2 -21673.433} C_VEL
LIN {X 0,Y 199.096,Z 382.219,A -85,B 0,C 180,E1 -21674.929,E2 -21674.929} C_VEL
LIN {X 0,Y 195.167,Z 385.411,A -85,B 0,C 180,E1 -21677.408,E2 -21677.408} C_VEL
LIN {X 0,Y 192.139,Z 387.369,A -85,B 0,C 180,E1 -21679.506,E2 -21679.506} C_VEL
LIN {X 0,Y 190.762,Z 388.512,A -85,B 0,C 180,E1 -21681.196,E2 -21681.196} C_VEL
LIN {X 0,Y 190.589,Z 388.828,A -85,B 0,C 180,E1 -21681.78,E2 -21681.78} C_VEL
LIN {X 0,Y 190.403,Z 390.472,A -85,B 0,C 180,E1 -21685.77,E2 -21685.77} C_VEL
LIN {X 0,Y 190.474,Z 390.775,A -85,B 0,C 180,E1 -21687.889,E2 -21687.889} C_VEL
LIN {X 0,Y 190.604,Z 390.669,A -85,B 0,C 180,E1 -21690.003,E2 -21690.003} C_VEL
LIN {X 0,Y 190.519,Z 390.109,A -85,B 0,C 180,E1 -21692.117,E2 -21692.117} C_VEL
LIN {X 0,Y 190.459,Z 388.771,A -85,B 0,C 180,E1 -21694.925,E2 -21694.925} C_VEL
LIN {X 0,Y 190.7,Z 385.978,A -85,B 0,C 180,E1 -21698.48,E2 -21698.48} C_VEL
LIN {X 0,Y 191.293,Z 382.404,A -85,B 0,C 180,E1 -21701.661,E2 -21701.661} C_VEL
LIN {X 0,Y 192.383,Z 377.717,A -85,B 0,C 180,E1 -21704.819,E2 -21704.819} C_VEL
LIN {X 0,Y 194.122,Z 371.786,A -85,B 0,C 180,E1 -21707.926,E2 -21707.926} C_VEL
LIN {X 0,Y 196.206,Z 364.374,A -85,B 0,C 180,E1 -21710.992,E2 -21710.992} C_VEL
LIN {X 0,Y 198.855,Z 355.191,A -85,B 0,C 180,E1 -21713.984,E2 -21713.984} C_VEL
LIN {X 0,Y 201.241,Z 346.733,A -85,B 0,C 180,E1 -21716.165,E2 -21716.165} C_VEL
LIN {X 0,Y 201.927,Z 336.147,A -85,B 0,C 180,E1 -21718.595,E2 -21718.595} C_VEL
LIN {X 0,Y 202.021,Z 325.946,A -85,B 0,C 180,E1 -21720.585,E2 -21720.585} C_VEL
LIN {X 0,Y 201.378,Z 314.356,A -85,B 0,C 180,E1 -21722.531,E2 -21722.531} C_VEL
LIN {X 0,Y 200.179,Z 304.348,A -85,B 0,C 180,E1 -21724.003,E2 -21724.003} C_VEL
LIN {X 0,Y 197.649,Z 292.07,A -85,B 0,C 180,E1 -21725.644,E2 -21725.644} C_VEL
LIN {X 0,Y 195.276,Z 282.719,A -85,B 0,C 180,E1 -21726.803,E2 -21726.803} C_VEL
LIN {X 0,Y 195.468,Z 280.671,A -85,B 0,C 180,E1 -21728.995,E2 -21728.995} C_VEL
LIN {X 0,Y 194.882,Z 276.953,A -85,B 0,C 180,E1 -21733.255,E2 -21733.255} C_VEL
LIN {X 0,Y 194.137,Z 273.092,A -85,B 0,C 180,E1 -21737.955,E2 -21737.955} C_VEL
LIN {X 0,Y 193.438,Z 269.22,A -85,B 0,C 180,E1 -21743.068,E2 -21743.068} C_VEL
LIN {X 0,Y 192.99,Z 266.628,A -85,B 0,C 180,E1 -21746.89,E2 -21746.89} C_VEL
LIN {X 0,Y 192.593,Z 264.493,A -85,B 0,C 180,E1 -21750.313,E2 -21750.313} C_VEL
LIN {X 0,Y 192.649,Z 264.487,A -85,B 0,C 180,E1 -21755.793,E2 -21755.793} C_VEL
LIN {X 0,Y 192.707,Z 264.481,A -85,B 0,C 180,E1 -21761.489,E2 -21761.489} C_VEL
LIN {X 0,Y 192.732,Z 264.479,A -85,B 0,C 180,E1 -21765.211,E2 -21765.211} C_VEL
LIN {X 0,Y 192.955,Z 264.452,A -85,B 0,C 180,E1 -21769.567,E2 -21769.567} C_VEL
LIN {X 0,Y 192.988,Z 264.446,A -85,B 0,C 180,E1 -21773.728,E2 -21773.728} C_VEL
LIN {X 0,Y 193.27,Z 264.412,A -85,B 0,C 180,E1 -21777.916,E2 -21777.916} C_VEL
LIN {X 0,Y 193.442,Z 264.384,A -85,B 0,C 180,E1 -21780,E2 -21780} C_VEL
LIN {X 0,Y 192.949,Z 264.446,A -85,B 0,C 180,E1 -21784.178,E2 -21784.178} C_VEL
LIN {X 0,Y 193.033,Z 264.438,A -85,B 0,C 180,E1 -21788.374,E2 -21788.374} C_VEL
LIN {X 0,Y 192.801,Z 264.469,A -85,B 0,C 180,E1 -21792.634,E2 -21792.634} C_VEL
LIN {X 0,Y 192.729,Z 264.479,A -85,B 0,C 180,E1 -21796.962,E2 -21796.962} C_VEL
LIN {X 0,Y 192.591,Z 264.495,A -85,B 0,C 180,E1 -21801.403,E2 -21801.403} C_VEL
LIN {X 0,Y 192.62,Z 264.487,A -85,B 0,C 180,E1 -21804.188,E2 -21804.188} C_VEL
LIN {X 0,Y 192.609,Z 264.489,A -85,B 0,C 180,E1 -21808.864,E2 -21808.864} C_VEL
LIN {X 0,Y 192.603,Z 264.489,A -85,B 0,C 180,E1 -21813.185,E2 -21813.185} C_VEL
LIN {X 0,Y 192.56,Z 264.5,A -85,B 0,C 180,E1 -21818.35,E2 -21818.35} C_VEL
LIN {X 0,Y 192.497,Z 264.505,A -85,B 0,C 180,E1 -21823.093,E2 -21823.093} C_VEL
LIN {X 0,Y 192.493,Z 264.507,A -85,B 0,C 180,E1 -21826.905,E2 -21826.905} C_VEL
LIN {X 0,Y 192.546,Z 264.501,A -85,B 0,C 180,E1 -21831.643,E2 -21831.643} C_VEL
LIN {X 0,Y 192.545,Z 264.502,A -85,B 0,C 180,E1 -21834.264,E2 -21834.264} C_VEL
LIN {X 0,Y 192.501,Z 264.919,A -85,B 0,C 180,E1 -21837.11,E2 -21837.11} C_VEL
LIN {X 0,Y 193.561,Z 267.772,A -85,B 0,C 180,E1 -21837.53,E2 -21837.53} C_VEL
LIN {X 0,Y 194.866,Z 270.268,A -85,B 0,C 180,E1 -21837.976,E2 -21837.976} C_VEL
LIN {X 0,Y 199.24,Z 280.643,A -85,B 0,C 180,E1 -21839.796,E2 -21839.796} C_VEL
LIN {X 0,Y 202.25,Z 290.129,A -85,B 0,C 180,E1 -21841.497,E2 -21841.497} C_VEL
LIN {X 0,Y 204.611,Z 300.572,A -85,B 0,C 180,E1 -21843.476,E2 -21843.476} C_VEL
LIN {X 0,Y 205.977,Z 310.162,A -85,B 0,C 180,E1 -21845.466,E2 -21845.466} C_VEL
LIN {X 0,Y 205.804,Z 313.174,A -85,B 0,C 180,E1 -21846.073,E2 -21846.073} C_VEL
LIN {X 0,Y 203.414,Z 323.521,A -85,B 0,C 180,E1 -21848.194,E2 -21848.194} C_VEL
LIN {X 0,Y 200.775,Z 332.871,A -85,B 0,C 180,E1 -21850.574,E2 -21850.574} C_VEL
LIN {X 0,Y 198.085,Z 341.864,A -85,B 0,C 180,E1 -21853.508,E2 -21853.508} C_VEL
LIN {X 0,Y 195.883,Z 349.107,A -85,B 0,C 180,E1 -21856.511,E2 -21856.511} C_VEL
LIN {X 0,Y 193.972,Z 354.924,A -85,B 0,C 180,E1 -21859.56,E2 -21859.56} C_VEL
LIN {X 0,Y 192.646,Z 359.502,A -85,B 0,C 180,E1 -21862.661,E2 -21862.661} C_VEL
LIN {X 0,Y 191.487,Z 363.013,A -85,B 0,C 180,E1 -21865.787,E2 -21865.787} C_VEL
LIN {X 0,Y 191.059,Z 364.799,A -85,B 0,C 180,E1 -21867.889,E2 -21867.889} C_VEL
LIN {X 0,Y 190.739,Z 367.099,A -85,B 0,C 180,E1 -21872.108,E2 -21872.108} C_VEL
LIN {X 0,Y 190.873,Z 367.869,A -85,B 0,C 180,E1 -21876.196,E2 -21876.196} C_VEL
LIN {X 0,Y 191.07,Z 367.638,A -85,B 0,C 180,E1 -21878.457,E2 -21878.457} C_VEL
LIN {X 0,Y 191.944,Z 366.046,A -85,B 0,C 180,E1 -21882.688,E2 -21882.688} C_VEL
LIN {X 0,Y 192.659,Z 364.635,A -85,B 0,C 180,E1 -21884.791,E2 -21884.791} C_VEL
LIN {X 0,Y 194.214,Z 361.706,A -85,B 0,C 180,E1 -21887.911,E2 -21887.911} C_VEL
LIN {X 0,Y 196.604,Z 356.695,A -85,B 0,C 180,E1 -21891.654,E2 -21891.654} C_VEL
LIN {X 0,Y 199.453,Z 350.576,A -85,B 0,C 180,E1 -21895.01,E2 -21895.01} C_VEL
LIN {X 0,Y 202.467,Z 343.595,A -85,B 0,C 180,E1 -21897.941,E2 -21897.941} C_VEL
LIN {X 0,Y 205.926,Z 334.831,A -85,B 0,C 180,E1 -21900.789,E2 -21900.789} C_VEL
LIN {X 0,Y 209.027,Z 325.826,A -85,B 0,C 180,E1 -21903.114,E2 -21903.114} C_VEL
LIN {X 0,Y 211.053,Z 319.403,A -85,B 0,C 180,E1 -21904.475,E2 -21904.475} C_VEL
LIN {X 0,Y 210.171,Z 310.978,A -85,B 0,C 180,E1 -21906.625,E2 -21906.625} C_VEL
LIN {X 0,Y 208.174,Z 300.764,A -85,B 0,C 180,E1 -21909.06,E2 -21909.06} C_VEL
LIN {X 0,Y 205.435,Z 291.668,A -85,B 0,C 180,E1 -21911.181,E2 -21911.181} C_VEL
LIN {X 0,Y 202.145,Z 283.476,A -85,B 0,C 180,E1 -21913.104,E2 -21913.104} C_VEL
LIN {X 0,Y 197.805,Z 274.963,A -85,B 0,C 180,E1 -21915.202,E2 -21915.202} C_VEL
LIN {X 0,Y 195.769,Z 271.459,A -85,B 0,C 180,E1 -21916.112,E2 -21916.112} C_VEL
LIN {X 0,Y 194.789,Z 270.105,A -85,B 0,C 180,E1 -21916.505,E2 -21916.505} C_VEL
LIN {X 0,Y 193.127,Z 267.217,A -85,B 0,C 180,E1 -21917.233,E2 -21917.233} C_VEL
LIN {X 0,Y 192.788,Z 266.023,A -85,B 0,C 180,E1 -21917.514,E2 -21917.514} C_VEL
LIN {X 0,Y 192.56,Z 264.497,A -85,B 0,C 180,E1 -21921.65,E2 -21921.65} C_VEL
LIN {X 0,Y 192.592,Z 264.492,A -85,B 0,C 180,E1 -21926.812,E2 -21926.812} C_VEL
LIN {X 0,Y 192.656,Z 264.483,A -85,B 0,C 180,E1 -21931.69,E2 -21931.69} C_VEL
LIN {X 0,Y 192.697,Z 264.483,A -85,B 0,C 180,E1 -21936.347,E2 -21936.347} C_VEL
LIN {X 0,Y 192.722,Z 264.477,A -85,B 0,C 180,E1 -21941.456,E2 -21941.456} C_VEL
LIN {X 0,Y 192.762,Z 264.475,A -85,B 0,C 180,E1 -21945.213,E2 -21945.213} C_VEL
LIN {X 0,Y 193.01,Z 264.444,A -85,B 0,C 180,E1 -21949.51,E2 -21949.51} C_VEL
LIN {X 0,Y 192.997,Z 264.444,A -85,B 0,C 180,E1 -21953.728,E2 -21953.728} C_VEL
LIN {X 0,Y 193.277,Z 264.409,A -85,B 0,C 180,E1 -21957.916,E2 -21957.916} C_VEL
LIN {X 0,Y 193.43,Z 264.39,A -85,B 0,C 180,E1 -21960,E2 -21960} C_VEL
LIN {X 0,Y 192.972,Z 264.446,A -85,B 0,C 180,E1 -21964.177,E2 -21964.177} C_VEL
LIN {X 0,Y 193.069,Z 264.435,A -85,B 0,C 180,E1 -21968.372,E2 -21968.372} C_VEL
LIN {X 0,Y 192.843,Z 264.461,A -85,B 0,C 180,E1 -21972.63,E2 -21972.63} C_VEL
LIN {X 0,Y 192.747,Z 264.472,A -85,B 0,C 180,E1 -21976.959,E2 -21976.959} C_VEL
LIN {X 0,Y 192.683,Z 264.475,A -85,B 0,C 180,E1 -21979.164,E2 -21979.164} C_VEL
LIN {X 0,Y 192.735,Z 265.015,A -85,B 0,C 180,E1 -21981.386,E2 -21981.386} C_VEL
LIN {X 0,Y 193.027,Z 266.456,A -85,B 0,C 180,E1 -21984.47,E2 -21984.47} C_VEL
LIN {X 0,Y 193.429,Z 269.008,A -85,B 0,C 180,E1 -21989.314,E2 -21989.314} C_VEL
LIN {X 0,Y 193.838,Z 271.496,A -85,B 0,C 180,E1 -21993.503,E2 -21993.503} C_VEL
LIN {X 0,Y 194.281,Z 274.425,A -85,B 0,C 180,E1 -21997.949,E2 -21997.949} C_VEL
LIN {X 0,Y 195.046,Z 278.228,A -85,B 0,C 180,E1 -22003.206,E2 -22003.206} C_VEL
LIN {X 0,Y 195.731,Z 281.928,A -85,B 0,C 180,E1 -22007.746,E2 -22007.746} C_VEL
LIN {X 0,Y 196.871,Z 285.116,A -85,B 0,C 180,E1 -22008.281,E2 -22008.281} C_VEL
LIN {X 0,Y 198.441,Z 287.632,A -85,B 0,C 180,E1 -22008.894,E2 -22008.894} C_VEL
LIN {X 0,Y 201.673,Z 295.621,A -85,B 0,C 180,E1 -22010.432,E2 -22010.432} C_VEL
LIN {X 0,Y 204.236,Z 306.732,A -85,B 0,C 180,E1 -22012.322,E2 -22012.322} C_VEL
LIN {X 0,Y 205.831,Z 317.35,A -85,B 0,C 180,E1 -22014.224,E2 -22014.224} C_VEL
LIN {X 0,Y 206.519,Z 328.289,A -85,B 0,C 180,E1 -22016.336,E2 -22016.336} C_VEL
LIN {X 0,Y 206.395,Z 338.789,A -85,B 0,C 180,E1 -22018.607,E2 -22018.607} C_VEL
LIN {X 0,Y 205.486,Z 347.942,A -85,B 0,C 180,E1 -22020.835,E2 -22020.835} C_VEL
LIN {X 0,Y 203.923,Z 353.548,A -85,B 0,C 180,E1 -22022.276,E2 -22022.276} C_VEL
LIN {X 0,Y 200.881,Z 361.544,A -85,B 0,C 180,E1 -22024.626,E2 -22024.626} C_VEL
LIN {X 0,Y 198.068,Z 368.808,A -85,B 0,C 180,E1 -22027.302,E2 -22027.302} C_VEL
LIN {X 0,Y 195.726,Z 374.771,A -85,B 0,C 180,E1 -22030.058,E2 -22030.058} C_VEL
LIN {X 0,Y 193.597,Z 380.022,A -85,B 0,C 180,E1 -22033.12,E2 -22033.12} C_VEL
LIN {X 0,Y 191.994,Z 384.12,A -85,B 0,C 180,E1 -22036.239,E2 -22036.239} C_VEL
LIN {X 0,Y 191.024,Z 387.182,A -85,B 0,C 180,E1 -22039.403,E2 -22039.403} C_VEL
LIN {X 0,Y 190.589,Z 388.828,A -85,B 0,C 180,E1 -22041.78,E2 -22041.78} C_VEL
LIN {X 0,Y 189.762,Z 389.709,A -85,B 0,C 180,E1 -22043.527,E2 -22043.527} C_VEL
LIN {X 0,Y 186.906,Z 390.431,A -85,B 0,C 180,E1 -22046.408,E2 -22046.408} C_VEL
LIN {X 0,Y 183.777,Z 390.246,A -85,B 0,C 180,E1 -22049.99,E2 -22049.99} C_VEL
LIN {X 0,Y 183.446,Z 389.908,A -85,B 0,C 180,E1 -22051.228,E2 -22051.228} C_VEL
LIN {X 0,Y 183.397,Z 388.423,A -85,B 0,C 180,E1 -22054.894,E2 -22054.894} C_VEL
LIN {X 0,Y 183.656,Z 385.475,A -85,B 0,C 180,E1 -22058.808,E2 -22058.808} C_VEL
LIN {X 0,Y 184.316,Z 381.877,A -85,B 0,C 180,E1 -22062.109,E2 -22062.109} C_VEL
LIN {X 0,Y 185.49,Z 377.161,A -85,B 0,C 180,E1 -22065.383,E2 -22065.383} C_VEL
LIN {X 0,Y 187.299,Z 371.198,A -85,B 0,C 180,E1 -22068.602,E2 -22068.602} C_VEL
LIN {X 0,Y 189.188,Z 365.133,A -85,B 0,C 180,E1 -22071.238,E2 -22071.238} C_VEL
LIN {X 0,Y 191.374,Z 357.833,A -85,B 0,C 180,E1 -22073.829,E2 -22073.829} C_VEL
LIN {X 0,Y 194.02,Z 349,A -85,B 0,C 180,E1 -22076.345,E2 -22076.345} C_VEL
LIN {X 0,Y 194.721,Z 344.887,A -85,B 0,C 180,E1 -22077.402,E2 -22077.402} C_VEL
LIN {X 0,Y 195.414,Z 334.207,A -85,B 0,C 180,E1 -22079.886,E2 -22079.886} C_VEL
LIN {X 0,Y 195.434,Z 323.352,A -85,B 0,C 180,E1 -22082.037,E2 -22082.037} C_VEL
LIN {X 0,Y 194.765,Z 312.42,A -85,B 0,C 180,E1 -22083.907,E2 -22083.907} C_VEL
LIN {X 0,Y 193.213,Z 301.391,A -85,B 0,C 180,E1 -22085.594,E2 -22085.594} C_VEL
LIN {X 0,Y 190.435,Z 289.127,A -85,B 0,C 180,E1 -22087.305,E2 -22087.305} C_VEL
LIN {X 0,Y 188.378,Z 282.265,A -85,B 0,C 180,E1 -22088.236,E2 -22088.236} C_VEL
LIN {X 0,Y 188.088,Z 279.347,A -85,B 0,C 180,E1 -22091.642,E2 -22091.642} C_VEL
LIN {X 0,Y 187.54,Z 276.312,A -85,B 0,C 180,E1 -22095.404,E2 -22095.404} C_VEL
LIN {X 0,Y 186.813,Z 272.618,A -85,B 0,C 180,E1 -22100.242,E2 -22100.242} C_VEL
LIN {X 0,Y 186.507,Z 270.679,A -85,B 0,C 180,E1 -22102.921,E2 -22102.921} C_VEL
LIN {X 0,Y 185.886,Z 267.369,A -85,B 0,C 180,E1 -22108.041,E2 -22108.041} C_VEL
LIN {X 0,Y 185.585,Z 265.365,A -85,B 0,C 180,E1 -22111.464,E2 -22111.464} C_VEL
LIN {X 0,Y 185.589,Z 265.366,A -85,B 0,C 180,E1 -22115.383,E2 -22115.383} C_VEL
LIN {X 0,Y 185.642,Z 265.36,A -85,B 0,C 180,E1 -22121.172,E2 -22121.172} C_VEL
LIN {X 0,Y 185.715,Z 265.353,A -85,B 0,C 180,E1 -22126.876,E2 -22126.876} C_VEL
LIN {X 0,Y 185.985,Z 265.319,A -85,B 0,C 180,E1 -22131.307,E2 -22131.307} C_VEL
LIN {X 0,Y 186.214,Z 265.29,A -85,B 0,C 180,E1 -22137.837,E2 -22137.837} C_VEL
LIN {X 0,Y 186.406,Z 265.26,A -85,B 0,C 180,E1 -22140,E2 -22140} C_VEL
LIN {X 0,Y 185.897,Z 265.325,A -85,B 0,C 180,E1 -22144.337,E2 -22144.337} C_VEL
LIN {X 0,Y 185.983,Z 265.316,A -85,B 0,C 180,E1 -22148.694,E2 -22148.694} C_VEL
LIN {X 0,Y 185.727,Z 265.349,A -85,B 0,C 180,E1 -22153.123,E2 -22153.123} C_VEL
LIN {X 0,Y 185.666,Z 265.357,A -85,B 0,C 180,E1 -22157.628,E2 -22157.628} C_VEL
LIN {X 0,Y 185.554,Z 265.372,A -85,B 0,C 180,E1 -22162.257,E2 -22162.257} C_VEL
LIN {X 0,Y 185.506,Z 265.378,A -85,B 0,C 180,E1 -22167.041,E2 -22167.041} C_VEL
LIN {X 0,Y 185.552,Z 265.368,A -85,B 0,C 180,E1 -22169.498,E2 -22169.498} C_VEL
LIN {X 0,Y 185.507,Z 265.378,A -85,B 0,C 180,E1 -22174.631,E2 -22174.631} C_VEL
LIN {X 0,Y 185.514,Z 265.374,A -85,B 0,C 180,E1 -22177.312,E2 -22177.312} C_VEL
LIN {X 0,Y 185.479,Z 265.381,A -85,B 0,C 180,E1 -22180.723,E2 -22180.723} C_VEL
LIN {X 0,Y 185.464,Z 265.382,A -85,B 0,C 180,E1 -22186.054,E2 -22186.054} C_VEL
LIN {X 0,Y 185.463,Z 265.383,A -85,B 0,C 180,E1 -22189.89,E2 -22189.89} C_VEL
LIN {X 0,Y 185.506,Z 265.378,A -85,B 0,C 180,E1 -22192.712,E2 -22192.712} C_VEL
LIN {X 0,Y 185.452,Z 265.536,A -85,B 0,C 180,E1 -22195.564,E2 -22195.564} C_VEL
LIN {X 0,Y 186.469,Z 268.474,A -85,B 0,C 180,E1 -22196.015,E2 -22196.015} C_VEL
LIN {X 0,Y 187.766,Z 270.509,A -85,B 0,C 180,E1 -22196.462,E2 -22196.462} C_VEL
LIN {X 0,Y 191.008,Z 277.486,A -85,B 0,C 180,E1 -22197.809,E2 -22197.809} C_VEL
LIN {X 0,Y 194.96,Z 288.4,A -85,B 0,C 180,E1 -22199.902,E2 -22199.902} C_VEL
LIN {X 0,Y 197.637,Z 299.194,A -85,B 0,C 180,E1 -22202.04,E2 -22202.04} C_VEL
LIN {X 0,Y 199.236,Z 309.467,A -85,B 0,C 180,E1 -22204.244,E2 -22204.244} C_VEL
LIN {X 0,Y 199.385,Z 314.019,A -85,B 0,C 180,E1 -22205.252,E2 -22205.252} C_VEL
LIN {X 0,Y 196.888,Z 324.293,A -85,B 0,C 180,E1 -22207.432,E2 -22207.432} C_VEL
LIN {X 0,Y 194.127,Z 333.567,A -85,B 0,C 180,E1 -22209.88,E2 -22209.88} C_VEL
LIN {X 0,Y 191.317,Z 342.511,A -85,B 0,C 180,E1 -22212.907,E2 -22212.907} C_VEL
LIN {X 0,Y 189.027,Z 349.714,A -85,B 0,C 180,E1 -22216.012,E2 -22216.012} C_VEL
LIN {X 0,Y 187.025,Z 355.498,A -85,B 0,C 180,E1 -22219.167,E2 -22219.167} C_VEL
LIN {X 0,Y 185.617,Z 360.046,A -85,B 0,C 180,E1 -22222.382,E2 -22222.382} C_VEL
LIN {X 0,Y 184.43,Z 363.526,A -85,B 0,C 180,E1 -22225.626,E2 -22225.626} C_VEL
LIN {X 0,Y 183.988,Z 365.284,A -85,B 0,C 180,E1 -22227.808,E2 -22227.808} C_VEL
LIN {X 0,Y 183.673,Z 367.557,A -85,B 0,C 180,E1 -22232.19,E2 -22232.19} C_VEL
LIN {X 0,Y 183.795,Z 368.29,A -85,B 0,C 180,E1 -22236.172,E2 -22236.172} C_VEL
LIN {X 0,Y 184.021,Z 368.048,A -85,B 0,C 180,E1 -22238.784,E2 -22238.784} C_VEL
LIN {X 0,Y 185.005,Z 366.429,A -85,B 0,C 180,E1 -22243.172,E2 -22243.172} C_VEL
LIN {X 0,Y 185.76,Z 364.991,A -85,B 0,C 180,E1 -22245.354,E2 -22245.354} C_VEL
LIN {X 0,Y 187.435,Z 362.035,A -85,B 0,C 180,E1 -22248.582,E2 -22248.582} C_VEL
LIN {X 0,Y 189.825,Z 357.31,A -85,B 0,C 180,E1 -22252.241,E2 -22252.241} C_VEL
LIN {X 0,Y 193.015,Z 350.84,A -85,B 0,C 180,E1 -22255.905,E2 -22255.905} C_VEL
LIN {X 0,Y 196.191,Z 343.802,A -85,B 0,C 180,E1 -22258.917,E2 -22258.917} C_VEL
LIN {X 0,Y 199.827,Z 334.992,A -85,B 0,C 180,E1 -22261.837,E2 -22261.837} C_VEL
LIN {X 0,Y 203.092,Z 325.934,A -85,B 0,C 180,E1 -22264.213,E2 -22264.213} C_VEL
LIN {X 0,Y 204.555,Z 321.718,A -85,B 0,C 180,E1 -22265.13,E2 -22265.13} C_VEL
LIN {X 0,Y 204.364,Z 316.188,A -85,B 0,C 180,E1 -22266.614,E2 -22266.614} C_VEL
LIN {X 0,Y 202.789,Z 306.133,A -85,B 0,C 180,E1 -22269.228,E2 -22269.228} C_VEL
LIN {X 0,Y 200.443,Z 296.87,A -85,B 0,C 180,E1 -22271.546,E2 -22271.546} C_VEL
LIN {X 0,Y 197.978,Z 289.878,A -85,B 0,C 180,E1 -22273.303,E2 -22273.303} C_VEL
LIN {X 0,Y 193.414,Z 280.039,A -85,B 0,C 180,E1 -22275.898,E2 -22275.898} C_VEL
LIN {X 0,Y 190.266,Z 274.759,A -85,B 0,C 180,E1 -22277.436,E2 -22277.436} C_VEL
LIN {X 0,Y 188.244,Z 271.174,A -85,B 0,C 180,E1 -22278.432,E2 -22278.432} C_VEL
LIN {X 0,Y 186.326,Z 268.544,A -85,B 0,C 180,E1 -22279.295,E2 -22279.295} C_VEL
LIN {X 0,Y 185.693,Z 266.642,A -85,B 0,C 180,E1 -22279.686,E2 -22279.686} C_VEL
LIN {X 0,Y 185.552,Z 265.588,A -85,B 0,C 180,E1 -22282.697,E2 -22282.697} C_VEL
LIN {X 0,Y 185.537,Z 265.373,A -85,B 0,C 180,E1 -22287.973,E2 -22287.973} C_VEL
LIN {X 0,Y 185.574,Z 265.37,A -85,B 0,C 180,E1 -22290.574,E2 -22290.574} C_VEL
LIN {X 0,Y 185.579,Z 265.367,A -85,B 0,C 180,E1 -22295.381,E2 -22295.381} C_VEL
LIN {X 0,Y 185.665,Z 265.357,A -85,B 0,C 180,E1 -22301.132,E2 -22301.132} C_VEL
LIN {X 0,Y 185.755,Z 265.346,A -85,B 0,C 180,E1 -22306.879,E2 -22306.879} C_VEL
LIN {X 0,Y 186.019,Z 265.313,A -85,B 0,C 180,E1 -22311.308,E2 -22311.308} C_VEL
LIN {X 0,Y 186.219,Z 265.288,A -85,B 0,C 180,E1 -22317.837,E2 -22317.837} C_VEL
LIN {X 0,Y 186.394,Z 265.266,A -85,B 0,C 180,E1 -22320,E2 -22320} C_VEL
LIN {X 0,Y 185.92,Z 265.325,A -85,B 0,C 180,E1 -22324.336,E2 -22324.336} C_VEL
LIN {X 0,Y 186.019,Z 265.312,A -85,B 0,C 180,E1 -22328.692,E2 -22328.692} C_VEL
LIN {X 0,Y 185.755,Z 265.344,A -85,B 0,C 180,E1 -22333.121,E2 -22333.121} C_VEL
LIN {X 0,Y 185.68,Z 265.354,A -85,B 0,C 180,E1 -22337.626,E2 -22337.626} C_VEL
LIN {X 0,Y 185.913,Z 267.058,A -85,B 0,C 180,E1 -22342.211,E2 -22342.211} C_VEL
LIN {X 0,Y 186.255,Z 269.323,A -85,B 0,C 180,E1 -22346.923,E2 -22346.923} C_VEL
LIN {X 0,Y 186.538,Z 270.924,A -85,B 0,C 180,E1 -22349.947,E2 -22349.947} C_VEL
LIN {X 0,Y 186.953,Z 273.497,A -85,B 0,C 180,E1 -22354.325,E2 -22354.325} C_VEL
LIN {X 0,Y 187.323,Z 275.877,A -85,B 0,C 180,E1 -22358.018,E2 -22358.018} C_VEL
LIN {X 0,Y 187.879,Z 278.875,A -85,B 0,C 180,E1 -22362.324,E2 -22362.324} C_VEL
LIN {X 0,Y 188.384,Z 281.234,A -85,B 0,C 180,E1 -22365.52,E2 -22365.52} C_VEL
LIN {X 0,Y 189.538,Z 284.432,A -85,B 0,C 180,E1 -22366.115,E2 -22366.115} C_VEL
LIN {X 0,Y 191.31,Z 287.171,A -85,B 0,C 180,E1 -22366.87,E2 -22366.87} C_VEL
LIN {X 0,Y 193.226,Z 291.181,A -85,B 0,C 180,E1 -22367.79,E2 -22367.79} C_VEL
LIN {X 0,Y 195.932,Z 297.892,A -85,B 0,C 180,E1 -22369.234,E2 -22369.234} C_VEL
LIN {X 0,Y 197.732,Z 304.82,A -85,B 0,C 180,E1 -22370.55,E2 -22370.55} C_VEL
LIN {X 0,Y 199.608,Z 316.963,A -85,B 0,C 180,E1 -22372.843,E2 -22372.843} C_VEL
LIN {X 0,Y 200.276,Z 326.866,A -85,B 0,C 180,E1 -22374.842,E2 -22374.842} C_VEL
LIN {X 0,Y 200.073,Z 338.56,A -85,B 0,C 180,E1 -22377.464,E2 -22377.464} C_VEL
LIN {X 0,Y 199.128,Z 347.783,A -85,B 0,C 180,E1 -22379.809,E2 -22379.809} C_VEL
LIN {X 0,Y 197.632,Z 353.368,A -85,B 0,C 180,E1 -22381.313,E2 -22381.313} C_VEL
LIN {X 0,Y 194.455,Z 361.322,A -85,B 0,C 180,E1 -22383.725,E2 -22383.725} C_VEL
LIN {X 0,Y 191.304,Z 369.048,A -85,B 0,C 180,E1 -22386.698,E2 -22386.698} C_VEL
LIN {X 0,Y 189.057,Z 374.481,A -85,B 0,C 180,E1 -22389.323,E2 -22389.323} C_VEL
LIN {X 0,Y 186.785,Z 379.699,A -85,B 0,C 180,E1 -22392.485,E2 -22392.485} C_VEL
LIN {X 0,Y 185.07,Z 383.773,A -85,B 0,C 180,E1 -22395.713,E2 -22395.713} C_VEL
LIN {X 0,Y 184.029,Z 386.815,A -85,B 0,C 180,E1 -22398.995,E2 -22398.995} C_VEL
LIN {X 0,Y 183.502,Z 388.554,A -85,B 0,C 180,E1 -22401.704,E2 -22401.704} C_VEL
LIN {X 0,Y 183.311,Z 390.06,A -85,B 0,C 180,E1 -22405.606,E2 -22405.606} C_VEL
LIN {X 0,Y 183.39,Z 390.353,A -85,B 0,C 180,E1 -22407.807,E2 -22407.807} C_VEL
LIN {X 0,Y 183.538,Z 390.228,A -85,B 0,C 180,E1 -22410.003,E2 -22410.003} C_VEL
LIN {X 0,Y 183.446,Z 389.908,A -85,B 0,C 180,E1 -22411.228,E2 -22411.228} C_VEL
LIN {X 0,Y 183.092,Z 389.543,A -85,B 0,C 180,E1 -22412.447,E2 -22412.447} C_VEL
LIN {X 0,Y 181.728,Z 388.699,A -85,B 0,C 180,E1 -22414.24,E2 -22414.24} C_VEL
LIN {X 0,Y 177.645,Z 385.692,A -85,B 0,C 180,E1 -22418.394,E2 -22418.394} C_VEL
LIN {X 0,Y 176.866,Z 383.965,A -85,B 0,C 180,E1 -22420.223,E2 -22420.223} C_VEL
LIN {X 0,Y 176.898,Z 383.321,A -85,B 0,C 180,E1 -22420.833,E2 -22420.833} C_VEL
LIN {X 0,Y 178.102,Z 378.3,A -85,B 0,C 180,E1 -22424.865,E2 -22424.865} C_VEL
LIN {X 0,Y 179.909,Z 372.761,A -85,B 0,C 180,E1 -22428.214,E2 -22428.214} C_VEL
LIN {X 0,Y 182.151,Z 365.865,A -85,B 0,C 180,E1 -22431.49,E2 -22431.49} C_VEL
LIN {X 0,Y 183.473,Z 361.346,A -85,B 0,C 180,E1 -22433.285,E2 -22433.285} C_VEL
LIN {X 0,Y 186.447,Z 352.049,A -85,B 0,C 180,E1 -22436.293,E2 -22436.293} C_VEL
LIN {X 0,Y 187.919,Z 346.286,A -85,B 0,C 180,E1 -22437.875,E2 -22437.875} C_VEL
LIN {X 0,Y 188.789,Z 335.652,A -85,B 0,C 180,E1 -22440.519,E2 -22440.519} C_VEL
LIN {X 0,Y 188.99,Z 324.059,A -85,B 0,C 180,E1 -22442.95,E2 -22442.95} C_VEL
LIN {X 0,Y 188.44,Z 313.547,A -85,B 0,C 180,E1 -22444.865,E2 -22444.865} C_VEL
LIN {X 0,Y 186.743,Z 301.128,A -85,B 0,C 180,E1 -22446.897,E2 -22446.897} C_VEL
LIN {X 0,Y 184.224,Z 289.896,A -85,B 0,C 180,E1 -22448.579,E2 -22448.579} C_VEL
LIN {X 0,Y 182.426,Z 285.239,A -85,B 0,C 180,E1 -22449.353,E2 -22449.353} C_VEL
LIN {X 0,Y 181.27,Z 281.76,A -85,B 0,C 180,E1 -22449.917,E2 -22449.917} C_VEL
LIN {X 0,Y 180.678,Z 278.172,A -85,B 0,C 180,E1 -22454.444,E2 -22454.444} C_VEL
LIN {X 0,Y 179.871,Z 274.177,A -85,B 0,C 180,E1 -22459.857,E2 -22459.857} C_VEL
LIN {X 0,Y 179.233,Z 270.438,A -85,B 0,C 180,E1 -22465.436,E2 -22465.436} C_VEL
LIN {X 0,Y 178.606,Z 266.636,A -85,B 0,C 180,E1 -22471.824,E2 -22471.824} C_VEL
LIN {X 0,Y 178.47,Z 266.252,A -85,B 0,C 180,E1 -22473.073,E2 -22473.073} C_VEL
LIN {X 0,Y 178.501,Z 266.25,A -85,B 0,C 180,E1 -22476.814,E2 -22476.814} C_VEL
LIN {X 0,Y 178.621,Z 266.236,A -85,B 0,C 180,E1 -22481.653,E2 -22481.653} C_VEL
LIN {X 0,Y 178.643,Z 266.235,A -85,B 0,C 180,E1 -22486.347,E2 -22486.347} C_VEL
LIN {X 0,Y 178.915,Z 266.2,A -85,B 0,C 180,E1 -22490.96,E2 -22490.96} C_VEL
LIN {X 0,Y 179.16,Z 266.168,A -85,B 0,C 180,E1 -22497.752,E2 -22497.752} C_VEL
LIN {X 0,Y 179.369,Z 266.137,A -85,B 0,C 180,E1 -22500,E2 -22500} C_VEL
LIN {X 0,Y 178.905,Z 266.199,A -85,B 0,C 180,E1 -22506.768,E2 -22506.768} C_VEL
LIN {X 0,Y 178.843,Z 266.203,A -85,B 0,C 180,E1 -22510.741,E2 -22510.741} C_VEL
LIN {X 0,Y 178.601,Z 266.235,A -85,B 0,C 180,E1 -22515.989,E2 -22515.989} C_VEL
LIN {X 0,Y 178.567,Z 266.236,A -85,B 0,C 180,E1 -22519.154,E2 -22519.154} C_VEL
LIN {X 0,Y 178.474,Z 266.249,A -85,B 0,C 180,E1 -22525.075,E2 -22525.075} C_VEL
LIN {X 0,Y 178.469,Z 266.255,A -85,B 0,C 180,E1 -22530.793,E2 -22530.793} C_VEL
LIN {X 0,Y 178.492,Z 266.249,A -85,B 0,C 180,E1 -22534.217,E2 -22534.217} C_VEL
LIN {X 0,Y 178.404,Z 266.261,A -85,B 0,C 180,E1 -22539.073,E2 -22539.073} C_VEL
LIN {X 0,Y 178.406,Z 266.262,A -85,B 0,C 180,E1 -22542.044,E2 -22542.044} C_VEL
LIN {X 0,Y 178.4,Z 266.261,A -85,B 0,C 180,E1 -22545.163,E2 -22545.163} C_VEL
LIN {X 0,Y 178.404,Z 266.263,A -85,B 0,C 180,E1 -22548.46,E2 -22548.46} C_VEL
LIN {X 0,Y 178.394,Z 266.31,A -85,B 0,C 180,E1 -22553.868,E2 -22553.868} C_VEL
LIN {X 0,Y 179.343,Z 269.051,A -85,B 0,C 180,E1 -22554.327,E2 -22554.327} C_VEL
LIN {X 0,Y 180.777,Z 271.221,A -85,B 0,C 180,E1 -22554.859,E2 -22554.859} C_VEL
LIN {X 0,Y 184.968,Z 279.708,A -85,B 0,C 180,E1 -22556.711,E2 -22556.711} C_VEL
LIN {X 0,Y 188.263,Z 288.85,A -85,B 0,C 180,E1 -22558.594,E2 -22558.594} C_VEL
LIN {X 0,Y 190.694,Z 297.828,A -85,B 0,C 180,E1 -22560.483,E2 -22560.483} C_VEL
LIN {X 0,Y 192.434,Z 307.84,A -85,B 0,C 180,E1 -22562.708,E2 -22562.708} C_VEL
LIN {X 0,Y 192.99,Z 314.866,A -85,B 0,C 180,E1 -22564.374,E2 -22564.374} C_VEL
LIN {X 0,Y 190.4,Z 325.064,A -85,B 0,C 180,E1 -22566.618,E2 -22566.618} C_VEL
LIN {X 0,Y 187.522,Z 334.256,A -85,B 0,C 180,E1 -22569.139,E2 -22569.139} C_VEL
LIN {X 0,Y 184.585,Z 343.156,A -85,B 0,C 180,E1 -22572.263,E2 -22572.263} C_VEL
LIN {X 0,Y 182.187,Z 350.32,A -85,B 0,C 180,E1 -22575.475,E2 -22575.475} C_VEL
LIN {X 0,Y 180.09,Z 356.068,A -85,B 0,C 180,E1 -22578.745,E2 -22578.745} C_VEL
LIN {X 0,Y 178.595,Z 360.585,A -85,B 0,C 180,E1 -22582.08,E2 -22582.08} C_VEL
LIN {X 0,Y 177.377,Z 364.038,A -85,B 0,C 180,E1 -22585.452,E2 -22585.452} C_VEL
LIN {X 0,Y 176.919,Z 365.769,A -85,B 0,C 180,E1 -22587.72,E2 -22587.72} C_VEL
LIN {X 0,Y 176.607,Z 368.016,A -85,B 0,C 180,E1 -22592.277,E2 -22592.277} C_VEL
LIN {X 0,Y 176.709,Z 368.702,A -85,B 0,C 180,E1 -22596.12,E2 -22596.12} C_VEL
LIN {X 0,Y 177.002,Z 368.456,A -85,B 0,C 180,E1 -22599.135,E2 -22599.135} C_VEL
LIN {X 0,Y 178.067,Z 366.81,A -85,B 0,C 180,E1 -22603.695,E2 -22603.695} C_VEL
LIN {X 0,Y 178.882,Z 365.348,A -85,B 0,C 180,E1 -22605.96,E2 -22605.96} C_VEL
LIN {X 0,Y 180.672,Z 362.363,A -85,B 0,C 180,E1 -22609.304,E2 -22609.304} C_VEL
LIN {X 0,Y 183.034,Z 357.963,A -85,B 0,C 180,E1 -22612.847,E2 -22612.847} C_VEL
LIN {X 0,Y 186.078,Z 352.105,A -85,B 0,C 180,E1 -22616.342,E2 -22616.342} C_VEL
LIN {X 0,Y 189.383,Z 345.307,A -85,B 0,C 180,E1 -22619.449,E2 -22619.449} C_VEL
LIN {X 0,Y 192.479,Z 338.343,A -85,B 0,C 180,E1 -22621.964,E2 -22621.964} C_VEL
LIN {X 0,Y 195.987,Z 329.379,A -85,B 0,C 180,E1 -22624.563,E2 -22624.563} C_VEL
LIN {X 0,Y 198.365,Z 322.864,A -85,B 0,C 180,E1 -22626.083,E2 -22626.083} C_VEL
LIN {X 0,Y 197.852,Z 315.527,A -85,B 0,C 180,E1 -22628.194,E2 -22628.194} C_VEL
LIN {X 0,Y 196.249,Z 305.86,A -85,B 0,C 180,E1 -22630.841,E2 -22630.841} C_VEL
LIN {X 0,Y 193.599,Z 296.153,A -85,B 0,C 180,E1 -22633.444,E2 -22633.444} C_VEL
LIN {X 0,Y 189.815,Z 287.015,A -85,B 0,C 180,E1 -22636.034,E2 -22636.034} C_VEL
LIN {X 0,Y 185.872,Z 279.579,A -85,B 0,C 180,E1 -22638.299,E2 -22638.299} C_VEL
LIN {X 0,Y 184.103,Z 276.379,A -85,B 0,C 180,E1 -22639.277,E2 -22639.277} C_VEL
LIN {X 0,Y 182.053,Z 272.987,A -85,B 0,C 180,E1 -22640.38,E2 -22640.38} C_VEL
LIN {X 0,Y 181.144,Z 271.764,A -85,B 0,C 180,E1 -22640.826,E2 -22640.826} C_VEL
LIN {X 0,Y 179.221,Z 269.126,A -85,B 0,C 180,E1 -22641.796,E2 -22641.796} C_VEL
LIN {X 0,Y 178.633,Z 267.235,A -85,B 0,C 180,E1 -22642.263,E2 -22642.263} C_VEL
LIN {X 0,Y 178.482,Z 266.248,A -85,B 0,C 180,E1 -22646.545,E2 -22646.545} C_VEL
LIN {X 0,Y 178.515,Z 266.244,A -85,B 0,C 180,E1 -22650.004,E2 -22650.004} C_VEL
LIN {X 0,Y 178.526,Z 266.247,A -85,B 0,C 180,E1 -22654.874,E2 -22654.874} C_VEL
LIN {X 0,Y 178.614,Z 266.237,A -85,B 0,C 180,E1 -22660.782,E2 -22660.782} C_VEL
LIN {X 0,Y 178.672,Z 266.227,A -85,B 0,C 180,E1 -22666.349,E2 -22666.349} C_VEL
LIN {X 0,Y 178.969,Z 266.19,A -85,B 0,C 180,E1 -22670.962,E2 -22670.962} C_VEL
LIN {X 0,Y 179.163,Z 266.167,A -85,B 0,C 180,E1 -22677.752,E2 -22677.752} C_VEL
LIN {X 0,Y 179.358,Z 266.143,A -85,B 0,C 180,E1 -22680,E2 -22680} C_VEL
LIN {X 0,Y 178.868,Z 266.203,A -85,B 0,C 180,E1 -22684.507,E2 -22684.507} C_VEL
LIN {X 0,Y 178.968,Z 266.19,A -85,B 0,C 180,E1 -22689.037,E2 -22689.037} C_VEL
LIN {X 0,Y 178.671,Z 266.228,A -85,B 0,C 180,E1 -22693.651,E2 -22693.651} C_VEL
LIN {X 0,Y 178.639,Z 266.352,A -85,B 0,C 180,E1 -22695.985,E2 -22695.985} C_VEL
LIN {X 0,Y 178.88,Z 268.122,A -85,B 0,C 180,E1 -22700.707,E2 -22700.707} C_VEL
LIN {X 0,Y 179.263,Z 270.29,A -85,B 0,C 180,E1 -22705.624,E2 -22705.624} C_VEL
LIN {X 0,Y 179.673,Z 272.84,A -85,B 0,C 180,E1 -22710.63,E2 -22710.63} C_VEL
LIN {X 0,Y 180.121,Z 275.869,A -85,B 0,C 180,E1 -22715.822,E2 -22715.822} C_VEL
LIN {X 0,Y 180.444,Z 277.782,A -85,B 0,C 180,E1 -22718.84,E2 -22718.84} C_VEL
LIN {X 0,Y 180.967,Z 280.627,A -85,B 0,C 180,E1 -22722.985,E2 -22722.985} C_VEL
LIN {X 0,Y 182.05,Z 283.621,A -85,B 0,C 180,E1 -22723.61,E2 -22723.61} C_VEL
LIN {X 0,Y 184.308,Z 286.964,A -85,B 0,C 180,E1 -22724.671,E2 -22724.671} C_VEL
LIN {X 0,Y 186.275,Z 290.957,A -85,B 0,C 180,E1 -22725.708,E2 -22725.708} C_VEL
LIN {X 0,Y 189.824,Z 298.802,A -85,B 0,C 180,E1 -22727.673,E2 -22727.673} C_VEL
LIN {X 0,Y 191.69,Z 305.08,A -85,B 0,C 180,E1 -22729.037,E2 -22729.037} C_VEL
LIN {X 0,Y 193.449,Z 317.045,A -85,B 0,C 180,E1 -22731.447,E2 -22731.447} C_VEL
LIN {X 0,Y 194.083,Z 327.944,A -85,B 0,C 180,E1 -22733.79,E2 -22733.79} C_VEL
LIN {X 0,Y 193.839,Z 338.136,A -85,B 0,C 180,E1 -22736.196,E2 -22736.196} C_VEL
LIN {X 0,Y 192.801,Z 347.623,A -85,B 0,C 180,E1 -22738.709,E2 -22738.709} C_VEL
LIN {X 0,Y 191.394,Z 353.189,A -85,B 0,C 180,E1 -22740.287,E2 -22740.287} C_VEL
LIN {X 0,Y 188.096,Z 361.101,A -85,B 0,C 180,E1 -22742.764,E2 -22742.764} C_VEL
LIN {X 0,Y 185.243,Z 367.679,A -85,B 0,C 180,E1 -22745.337,E2 -22745.337} C_VEL
LIN {X 0,Y 182.421,Z 374.189,A -85,B 0,C 180,E1 -22748.535,E2 -22748.535} C_VEL
LIN {X 0,Y 180.002,Z 379.375,A -85,B 0,C 180,E1 -22751.803,E2 -22751.803} C_VEL
LIN {X 0,Y 178.146,Z 383.423,A -85,B 0,C 180,E1 -22755.145,E2 -22755.145} C_VEL
LIN {X 0,Y 177.021,Z 386.446,A -85,B 0,C 180,E1 -22758.554,E2 -22758.554} C_VEL
LIN {X 0,Y 176.548,Z 387.917,A -85,B 0,C 180,E1 -22760.841,E2 -22760.841} C_VEL
LIN {X 0,Y 176.261,Z 389.65,A -85,B 0,C 180,E1 -22765.429,E2 -22765.429} C_VEL
LIN {X 0,Y 176.306,Z 389.932,A -85,B 0,C 180,E1 -22767.719,E2 -22767.719} C_VEL
LIN {X 0,Y 176.472,Z 389.786,A -85,B 0,C 180,E1 -22770.003,E2 -22770.003} C_VEL
LIN {X 0,Y 176.35,Z 389.2,A -85,B 0,C 180,E1 -22772.287,E2 -22772.287} C_VEL
LIN {X 0,Y 176.327,Z 388.087,A -85,B 0,C 180,E1 -22774.833,E2 -22774.833} C_VEL
LIN {X 0,Y 176.61,Z 384.971,A -85,B 0,C 180,E1 -22779.162,E2 -22779.162} C_VEL
LIN {X 0,Y 176.898,Z 383.321,A -85,B 0,C 180,E1 -22780.833,E2 -22780.833} C_VEL
LIN {X 0,Y 176.654,Z 381.308,A -85,B 0,C 180,E1 -22782.633,E2 -22782.633} C_VEL
LIN {X 0,Y 174.771,Z 377.496,A -85,B 0,C 180,E1 -22785.567,E2 -22785.567} C_VEL
LIN {X 0,Y 173.337,Z 373.057,A -85,B 0,C 180,E1 -22788.453,E2 -22788.453} C_VEL
LIN {X 0,Y 173.785,Z 370.005,A -85,B 0,C 180,E1 -22790.117,E2 -22790.117} C_VEL
LIN {X 0,Y 175.337,Z 365.609,A -85,B 0,C 180,E1 -22792.194,E2 -22792.194} C_VEL
LIN {X 0,Y 177.321,Z 359.617,A -85,B 0,C 180,E1 -22794.596,E2 -22794.596} C_VEL
LIN {X 0,Y 180.067,Z 351.367,A -85,B 0,C 180,E1 -22797.3,E2 -22797.3} C_VEL
LIN {X 0,Y 181.255,Z 346.559,A -85,B 0,C 180,E1 -22798.678,E2 -22798.678} C_VEL
LIN {X 0,Y 182.219,Z 336.686,A -85,B 0,C 180,E1 -22801.282,E2 -22801.282} C_VEL
LIN {X 0,Y 182.596,Z 326.582,A -85,B 0,C 180,E1 -22803.561,E2 -22803.561} C_VEL
LIN {X 0,Y 182.162,Z 314.703,A -85,B 0,C 180,E1 -22805.884,E2 -22805.884} C_VEL
LIN {X 0,Y 180.659,Z 302.438,A -85,B 0,C 180,E1 -22808.023,E2 -22808.023} C_VEL
LIN {X 0,Y 178.412,Z 292.413,A -85,B 0,C 180,E1 -22809.69,E2 -22809.69} C_VEL
LIN {X 0,Y 175.986,Z 285.957,A -85,B 0,C 180,E1 -22810.872,E2 -22810.872} C_VEL
LIN {X 0,Y 174.366,Z 282.834,A -85,B 0,C 180,E1 -22811.543,E2 -22811.543} C_VEL
LIN {X 0,Y 174.019,Z 281.27,A -85,B 0,C 180,E1 -22811.765,E2 -22811.765} C_VEL
LIN {X 0,Y 173.282,Z 277.489,A -85,B 0,C 180,E1 -22816.895,E2 -22816.895} C_VEL
LIN {X 0,Y 172.803,Z 274.935,A -85,B 0,C 180,E1 -22820.606,E2 -22820.606} C_VEL
LIN {X 0,Y 172.289,Z 272.013,A -85,B 0,C 180,E1 -22825.174,E2 -22825.174} C_VEL
LIN {X 0,Y 171.735,Z 268.837,A -85,B 0,C 180,E1 -22830.588,E2 -22830.588} C_VEL
LIN {X 0,Y 171.437,Z 267.128,A -85,B 0,C 180,E1 -22833.918,E2 -22833.918} C_VEL
LIN {X 0,Y 171.453,Z 267.128,A -85,B 0,C 180,E1 -22838.351,E2 -22838.351} C_VEL
LIN {X 0,Y 171.554,Z 267.116,A -85,B 0,C 180,E1 -22840.869,E2 -22840.869} C_VEL
LIN {X 0,Y 171.558,Z 267.117,A -85,B 0,C 180,E1 -22845.771,E2 -22845.771} C_VEL
LIN {X 0,Y 171.853,Z 267.08,A -85,B 0,C 180,E1 -22850.585,E2 -22850.585} C_VEL
LIN {X 0,Y 171.82,Z 267.081,A -85,B 0,C 180,E1 -22855.308,E2 -22855.308} C_VEL
LIN {X 0,Y 172.332,Z 267.013,A -85,B 0,C 180,E1 -22860,E2 -22860} C_VEL
LIN {X 0,Y 171.868,Z 267.077,A -85,B 0,C 180,E1 -22867.047,E2 -22867.047} C_VEL
LIN {X 0,Y 171.777,Z 267.084,A -85,B 0,C 180,E1 -22870.894,E2 -22870.894} C_VEL
LIN {X 0,Y 171.531,Z 267.117,A -85,B 0,C 180,E1 -22876.667,E2 -22876.667} C_VEL
LIN {X 0,Y 171.491,Z 267.116,A -85,B 0,C 180,E1 -22879.501,E2 -22879.501} C_VEL
LIN {X 0,Y 171.412,Z 267.13,A -85,B 0,C 180,E1 -22885.568,E2 -22885.568} C_VEL
LIN {X 0,Y 171.426,Z 267.13,A -85,B 0,C 180,E1 -22890.571,E2 -22890.571} C_VEL
LIN {X 0,Y 171.401,Z 267.135,A -85,B 0,C 180,E1 -22895.033,E2 -22895.033} C_VEL
LIN {X 0,Y 171.366,Z 267.139,A -85,B 0,C 180,E1 -22898.806,E2 -22898.806} C_VEL
LIN {X 0,Y 171.328,Z 267.145,A -85,B 0,C 180,E1 -22904.216,E2 -22904.216} C_VEL
LIN {X 0,Y 171.337,Z 267.144,A -85,B 0,C 180,E1 -22908.978,E2 -22908.978} C_VEL
LIN {X 0,Y 171.381,Z 267.2,A -85,B 0,C 180,E1 -22912.009,E2 -22912.009} C_VEL
LIN {X 0,Y 172.33,Z 269.91,A -85,B 0,C 180,E1 -22912.511,E2 -22912.511} C_VEL
LIN {X 0,Y 173.879,Z 272.133,A -85,B 0,C 180,E1 -22913.131,E2 -22913.131} C_VEL
LIN {X 0,Y 178.792,Z 281.538,A -85,B 0,C 180,E1 -22915.442,E2 -22915.442} C_VEL
LIN {X 0,Y 182.585,Z 292.393,A -85,B 0,C 180,E1 -22917.868,E2 -22917.868} C_VEL
LIN {X 0,Y 184.912,Z 302.045,A -85,B 0,C 180,E1 -22920.073,E2 -22920.073} C_VEL
LIN {X 0,Y 186.293,Z 311.734,A -85,B 0,C 180,E1 -22922.406,E2 -22922.406} C_VEL
LIN {X 0,Y 186.595,Z 315.719,A -85,B 0,C 180,E1 -22923.428,E2 -22923.428} C_VEL
LIN {X 0,Y 183.956,Z 325.826,A -85,B 0,C 180,E1 -22925.748,E2 -22925.748} C_VEL
LIN {X 0,Y 180.959,Z 334.944,A -85,B 0,C 180,E1 -22928.345,E2 -22928.345} C_VEL
LIN {X 0,Y 177.885,Z 343.8,A -85,B 0,C 180,E1 -22931.571,E2 -22931.571} C_VEL
LIN {X 0,Y 175.364,Z 350.927,A -85,B 0,C 180,E1 -22934.897,E2 -22934.897} C_VEL
LIN {X 0,Y 173.166,Z 356.633,A -85,B 0,C 180,E1 -22938.288,E2 -22938.288} C_VEL
LIN {X 0,Y 171.578,Z 361.119,A -85,B 0,C 180,E1 -22941.754,E2 -22941.754} C_VEL
LIN {X 0,Y 170.328,Z 364.547,A -85,B 0,C 180,E1 -22945.263,E2 -22945.263} C_VEL
LIN {X 0,Y 169.853,Z 366.254,A -85,B 0,C 180,E1 -22947.625,E2 -22947.625} C_VEL
LIN {X 0,Y 169.543,Z 368.474,A -85,B 0,C 180,E1 -22952.372,E2 -22952.372} C_VEL
LIN {X 0,Y 169.647,Z 369.117,A -85,B 0,C 180,E1 -22956.14,E2 -22956.14} C_VEL
LIN {X 0,Y 169.962,Z 368.865,A -85,B 0,C 180,E1 -22959.517,E2 -22959.517} C_VEL
LIN {X 0,Y 170.453,Z 368.222,A -85,B 0,C 180,E1 -22961.894,E2 -22961.894} C_VEL
LIN {X 0,Y 171.13,Z 367.189,A -85,B 0,C 180,E1 -22964.261,E2 -22964.261} C_VEL
LIN {X 0,Y 172.03,Z 365.704,A -85,B 0,C 180,E1 -22966.613,E2 -22966.613} C_VEL
LIN {X 0,Y 173.943,Z 362.691,A -85,B 0,C 180,E1 -22970.082,E2 -22970.082} C_VEL
LIN {X 0,Y 176.322,Z 358.55,A -85,B 0,C 180,E1 -22973.543,E2 -22973.543} C_VEL
LIN {X 0,Y 179.726,Z 352.368,A -85,B 0,C 180,E1 -22977.349,E2 -22977.349} C_VEL
LIN {X 0,Y 183.199,Z 345.534,A -85,B 0,C 180,E1 -22980.547,E2 -22980.547} C_VEL
LIN {X 0,Y 187.15,Z 336.939,A -85,B 0,C 180,E1 -22983.631,E2 -22983.631} C_VEL
LIN {X 0,Y 190.687,Z 328.1,A -85,B 0,C 180,E1 -22986.132,E2 -22986.132} C_VEL
LIN {X 0,Y 192.087,Z 324.014,A -85,B 0,C 180,E1 -22987.131,E2 -22987.131} C_VEL
LIN {X 0,Y 191.368,Z 314.749,A -85,B 0,C 180,E1 -22989.947,E2 -22989.947} C_VEL
LIN {X 0,Y 189.976,Z 306.728,A -85,B 0,C 180,E1 -22992.278,E2 -22992.278} C_VEL
LIN {X 0,Y 187.731,Z 298.585,A -85,B 0,C 180,E1 -22994.659,E2 -22994.659} C_VEL
LIN {X 0,Y 184.187,Z 289.754,A -85,B 0,C 180,E1 -22997.368,E2 -22997.368} C_VEL
LIN {X 0,Y 179.645,Z 281.152,A -85,B 0,C 180,E1 -23000.253,E2 -23000.253} C_VEL
LIN {X 0,Y 177.408,Z 277.378,A -85,B 0,C 180,E1 -23001.601,E2 -23001.601} C_VEL
LIN {X 0,Y 175.217,Z 273.882,A -85,B 0,C 180,E1 -23002.904,E2 -23002.904} C_VEL
LIN {X 0,Y 174.629,Z 272.811,A -85,B 0,C 180,E1 -23003.262,E2 -23003.262} C_VEL
LIN {X 0,Y 172.404,Z 270.25,A -85,B 0,C 180,E1 -23004.477,E2 -23004.477} C_VEL
LIN {X 0,Y 171.53,Z 267.895,A -85,B 0,C 180,E1 -23005.151,E2 -23005.151} C_VEL
LIN {X 0,Y 171.411,Z 267.183,A -85,B 0,C 180,E1 -23007.79,E2 -23007.79} C_VEL
LIN {X 0,Y 171.441,Z 267.129,A -85,B 0,C 180,E1 -23010.532,E2 -23010.532} C_VEL
LIN {X 0,Y 171.449,Z 267.128,A -85,B 0,C 180,E1 -23015.8,E2 -23015.8} C_VEL
LIN {X 0,Y 171.57,Z 267.114,A -85,B 0,C 180,E1 -23020.87,E2 -23020.87} C_VEL
LIN {X 0,Y 171.585,Z 267.11,A -85,B 0,C 180,E1 -23025.773,E2 -23025.773} C_VEL
LIN {X 0,Y 171.9,Z 267.071,A -85,B 0,C 180,E1 -23030.587,E2 -23030.587} C_VEL
LIN {X 0,Y 171.827,Z 267.081,A -85,B 0,C 180,E1 -23035.307,E2 -23035.307} C_VEL
LIN {X 0,Y 172.321,Z 267.019,A -85,B 0,C 180,E1 -23040,E2 -23040} C_VEL
LIN {X 0,Y 171.818,Z 267.081,A -85,B 0,C 180,E1 -23044.692,E2 -23044.692} C_VEL
LIN {X 0,Y 171.9,Z 267.072,A -85,B 0,C 180,E1 -23049.412,E2 -23049.412} C_VEL
LIN {X 0,Y 171.737,Z 267.093,A -85,B 0,C 180,E1 -23051.807,E2 -23051.807} C_VEL
LIN {X 0,Y 171.776,Z 268.305,A -85,B 0,C 180,E1 -23056.642,E2 -23056.642} C_VEL
LIN {X 0,Y 172.022,Z 270.155,A -85,B 0,C 180,E1 -23061.573,E2 -23061.573} C_VEL
LIN {X 0,Y 172.384,Z 272.385,A -85,B 0,C 180,E1 -23066.645,E2 -23066.645} C_VEL
LIN {X 0,Y 172.793,Z 275.08,A -85,B 0,C 180,E1 -23071.921,E2 -23071.921} C_VEL
LIN {X 0,Y 173.16,Z 277.254,A -85,B 0,C 180,E1 -23075.741,E2 -23075.741} C_VEL
LIN {X 0,Y 173.571,Z 279.939,A -85,B 0,C 180,E1 -23080.084,E2 -23080.084} C_VEL
LIN {X 0,Y 174.702,Z 283.027,A -85,B 0,C 180,E1 -23080.822,E2 -23080.822} C_VEL
LIN {X 0,Y 177.098,Z 286.489,A -85,B 0,C 180,E1 -23082.087,E2 -23082.087} C_VEL
LIN {X 0,Y 179.027,Z 290.391,A -85,B 0,C 180,E1 -23083.229,E2 -23083.229} C_VEL
LIN {X 0,Y 180.114,Z 292.194,A -85,B 0,C 180,E1 -23083.815,E2 -23083.815} C_VEL
LIN {X 0,Y 182.673,Z 297.738,A -85,B 0,C 180,E1 -23085.378,E2 -23085.378} C_VEL
LIN {X 0,Y 185.286,Z 304.233,A -85,B 0,C 180,E1 -23087.116,E2 -23087.116} C_VEL
LIN {X 0,Y 186.808,Z 311.766,A -85,B 0,C 180,E1 -23088.801,E2 -23088.801} C_VEL
LIN {X 0,Y 187.875,Z 323.619,A -85,B 0,C 180,E1 -23091.42,E2 -23091.42} C_VEL
LIN {X 0,Y 187.89,Z 332.771,A -85,B 0,C 180,E1 -23093.577,E2 -23093.577} C_VEL
LIN {X 0,Y 187.228,Z 342.505,A -85,B 0,C 180,E1 -23096.12,E2 -23096.12} C_VEL
LIN {X 0,Y 185.782,Z 351.217,A -85,B 0,C 180,E1 -23098.662,E2 -23098.662} C_VEL
LIN {X 0,Y 183.127,Z 357.894,A -85,B 0,C 180,E1 -23100.708,E2 -23100.708} C_VEL
LIN {X 0,Y 179.359,Z 366.182,A -85,B 0,C 180,E1 -23103.848,E2 -23103.848} C_VEL
LIN {X 0,Y 176.277,Z 372.888,A -85,B 0,C 180,E1 -23107.129,E2 -23107.129} C_VEL
LIN {X 0,Y 173.246,Z 379.048,A -85,B 0,C 180,E1 -23111.066,E2 -23111.066} C_VEL
LIN {X 0,Y 171.254,Z 383.072,A -85,B 0,C 180,E1 -23114.533,E2 -23114.533} C_VEL
LIN {X 0,Y 170.037,Z 386.076,A -85,B 0,C 180,E1 -23118.077,E2 -23118.077} C_VEL
LIN {X 0,Y 169.237,Z 388.576,A -85,B 0,C 180,E1 -23122.847,E2 -23122.847} C_VEL
LIN {X 0,Y 169.163,Z 389.324,A -85,B 0,C 180,E1 -23125.632,E2 -23125.632} C_VEL
LIN {X 0,Y 169.407,Z 389.343,A -85,B 0,C 180,E1 -23130.003,E2 -23130.003} C_VEL
LIN {X 0,Y 169.268,Z 388.745,A -85,B 0,C 180,E1 -23132.383,E2 -23132.383} C_VEL
LIN {X 0,Y 169.243,Z 387.749,A -85,B 0,C 180,E1 -23134.768,E2 -23134.768} C_VEL
LIN {X 0,Y 169.276,Z 386.341,A -85,B 0,C 180,E1 -23137.158,E2 -23137.158} C_VEL
LIN {X 0,Y 169.82,Z 383.134,A -85,B 0,C 180,E1 -23140.973,E2 -23140.973} C_VEL
LIN {X 0,Y 170.735,Z 379.362,A -85,B 0,C 180,E1 -23144.302,E2 -23144.302} C_VEL
LIN {X 0,Y 172.777,Z 373.21,A -85,B 0,C 180,E1 -23148.379,E2 -23148.379} C_VEL
LIN {X 0,Y 173.785,Z 370.005,A -85,B 0,C 180,E1 -23150.117,E2 -23150.117} C_VEL
LIN {X 0,Y 173.909,Z 367.887,A -85,B 0,C 180,E1 -23151.22,E2 -23151.22} C_VEL
LIN {X 0,Y 172.363,Z 364.371,A -85,B 0,C 180,E1 -23153.061,E2 -23153.061} C_VEL
LIN {X 0,Y 170.906,Z 360.654,A -85,B 0,C 180,E1 -23154.885,E2 -23154.885} C_VEL
LIN {X 0,Y 171.171,Z 358.102,A -85,B 0,C 180,E1 -23155.922,E2 -23155.922} C_VEL
LIN {X 0,Y 174.288,Z 348.839,A -85,B 0,C 180,E1 -23158.943,E2 -23158.943} C_VEL
LIN {X 0,Y 175.55,Z 338.992,A -85,B 0,C 180,E1 -23161.748,E2 -23161.748} C_VEL
LIN {X 0,Y 176.156,Z 328.751,A -85,B 0,C 180,E1 -23164.248,E2 -23164.248} C_VEL
LIN {X 0,Y 176.065,Z 317.919,A -85,B 0,C 180,E1 -23166.552,E2 -23166.552} C_VEL
LIN {X 0,Y 174.913,Z 305.974,A -85,B 0,C 180,E1 -23168.841,E2 -23168.841} C_VEL
LIN {X 0,Y 173.057,Z 296.093,A -85,B 0,C 180,E1 -23170.614,E2 -23170.614} C_VEL
LIN {X 0,Y 170.671,Z 289.684,A -85,B 0,C 180,E1 -23171.945,E2 -23171.945} C_VEL
LIN {X 0,Y 168.56,Z 285.167,A -85,B 0,C 180,E1 -23172.952,E2 -23172.952} C_VEL
LIN {X 0,Y 166.996,Z 281.96,A -85,B 0,C 180,E1 -23173.681,E2 -23173.681} C_VEL
LIN {X 0,Y 166.718,Z 280.711,A -85,B 0,C 180,E1 -23173.903,E2 -23173.903} C_VEL
LIN {X 0,Y 165.943,Z 276.8,A -85,B 0,C 180,E1 -23179.675,E2 -23179.675} C_VEL
LIN {X 0,Y 165.437,Z 274.184,A -85,B 0,C 180,E1 -23183.823,E2 -23183.823} C_VEL
LIN {X 0,Y 164.895,Z 271.059,A -85,B 0,C 180,E1 -23189.239,E2 -23189.239} C_VEL
LIN {X 0,Y 164.407,Z 268.004,A -85,B 0,C 180,E1 -23195.368,E2 -23195.368} C_VEL
LIN {X 0,Y 164.448,Z 268.001,A -85,B 0,C 180,E1 -23200.097,E2 -23200.097} C_VEL
LIN {X 0,Y 164.488,Z 267.998,A -85,B 0,C 180,E1 -23205.146,E2 -23205.146} C_VEL
LIN {X 0,Y 164.774,Z 267.963,A -85,B 0,C 180,E1 -23210.177,E2 -23210.177} C_VEL
LIN {X 0,Y 164.836,Z 267.949,A -85,B 0,C 180,E1 -23212.651,E2 -23212.651} C_VEL
LIN {X 0,Y 165.055,Z 267.923,A -85,B 0,C 180,E1 -23217.56,E2 -23217.56} C_VEL
LIN {X 0,Y 165.295,Z 267.889,A -85,B 0,C 180,E1 -23220,E2 -23220} C_VEL
LIN {X 0,Y 164.829,Z 267.954,A -85,B 0,C 180,E1 -23227.349,E2 -23227.349} C_VEL
LIN {X 0,Y 164.711,Z 267.965,A -85,B 0,C 180,E1 -23231.058,E2 -23231.058} C_VEL
LIN {X 0,Y 164.451,Z 268,A -85,B 0,C 180,E1 -23237.407,E2 -23237.407} C_VEL
LIN {X 0,Y 164.429,Z 267.995,A -85,B 0,C 180,E1 -23239.995,E2 -23239.995} C_VEL
LIN {X 0,Y 164.347,Z 268.012,A -85,B 0,C 180,E1 -23246.093,E2 -23246.093} C_VEL
LIN {X 0,Y 164.366,Z 268.011,A -85,B 0,C 180,E1 -23251.216,E2 -23251.216} C_VEL
LIN {X 0,Y 164.303,Z 268.015,A -85,B 0,C 180,E1 -23256.788,E2 -23256.788} C_VEL
LIN {X 0,Y 164.299,Z 268.017,A -85,B 0,C 180,E1 -23259.914,E2 -23259.914} C_VEL
LIN {X 0,Y 164.288,Z 268.019,A -85,B 0,C 180,E1 -23263.34,E2 -23263.34} C_VEL
LIN {X 0,Y 164.281,Z 268.022,A -85,B 0,C 180,E1 -23268.461,E2 -23268.461} C_VEL
LIN {X 0,Y 164.3,Z 268.181,A -85,B 0,C 180,E1 -23269.921,E2 -23269.921} C_VEL
LIN {X 0,Y 165.302,Z 270.907,A -85,B 0,C 180,E1 -23270.491,E2 -23270.491} C_VEL
LIN {X 0,Y 167.028,Z 273.116,A -85,B 0,C 180,E1 -23271.235,E2 -23271.235} C_VEL
LIN {X 0,Y 168.909,Z 276.369,A -85,B 0,C 180,E1 -23272.157,E2 -23272.157} C_VEL
LIN {X 0,Y 173.632,Z 285.845,A -85,B 0,C 180,E1 -23274.692,E2 -23274.692} C_VEL
LIN {X 0,Y 176.979,Z 296.325,A -85,B 0,C 180,E1 -23277.232,E2 -23277.232} C_VEL
LIN {X 0,Y 178.781,Z 304.581,A -85,B 0,C 180,E1 -23279.263,E2 -23279.263} C_VEL
LIN {X 0,Y 179.975,Z 314.137,A -85,B 0,C 180,E1 -23281.734,E2 -23281.734} C_VEL
LIN {X 0,Y 180.073,Z 317.784,A -85,B 0,C 180,E1 -23282.701,E2 -23282.701} C_VEL
LIN {X 0,Y 177.56,Z 326.574,A -85,B 0,C 180,E1 -23284.814,E2 -23284.814} C_VEL
LIN {X 0,Y 174.435,Z 335.631,A -85,B 0,C 180,E1 -23287.492,E2 -23287.492} C_VEL
LIN {X 0,Y 171.192,Z 344.446,A -85,B 0,C 180,E1 -23290.823,E2 -23290.823} C_VEL
LIN {X 0,Y 168.56,Z 351.53,A -85,B 0,C 180,E1 -23294.272,E2 -23294.272} C_VEL
LIN {X 0,Y 166.256,Z 357.194,A -85,B 0,C 180,E1 -23297.794,E2 -23297.794} C_VEL
LIN {X 0,Y 164.572,Z 361.65,A -85,B 0,C 180,E1 -23301.4,E2 -23301.4} C_VEL
LIN {X 0,Y 163.282,Z 365.051,A -85,B 0,C 180,E1 -23305.058,E2 -23305.058} C_VEL
LIN {X 0,Y 162.525,Z 368.029,A -85,B 0,C 180,E1 -23309.996,E2 -23309.996} C_VEL
LIN {X 0,Y 162.456,Z 368.934,A -85,B 0,C 180,E1 -23312.476,E2 -23312.476} C_VEL
LIN {X 0,Y 162.55,Z 369.526,A -85,B 0,C 180,E1 -23316.046,E2 -23316.046} C_VEL
LIN {X 0,Y 162.942,Z 369.275,A -85,B 0,C 180,E1 -23319.931,E2 -23319.931} C_VEL
LIN {X 0,Y 163.471,Z 368.619,A -85,B 0,C 180,E1 -23322.41,E2 -23322.41} C_VEL
LIN {X 0,Y 164.218,Z 367.564,A -85,B 0,C 180,E1 -23324.875,E2 -23324.875} C_VEL
LIN {X 0,Y 165.203,Z 366.061,A -85,B 0,C 180,E1 -23327.321,E2 -23327.321} C_VEL
LIN {X 0,Y 167.254,Z 363.019,A -85,B 0,C 180,E1 -23330.923,E2 -23330.923} C_VEL
LIN {X 0,Y 169.752,Z 358.921,A -85,B 0,C 180,E1 -23334.453,E2 -23334.453} C_VEL
LIN {X 0,Y 173.423,Z 352.633,A -85,B 0,C 180,E1 -23338.432,E2 -23338.432} C_VEL
LIN {X 0,Y 177.091,Z 345.759,A -85,B 0,C 180,E1 -23341.72,E2 -23341.72} C_VEL
LIN {X 0,Y 181.237,Z 337.104,A -85,B 0,C 180,E1 -23344.884,E2 -23344.884} C_VEL
LIN {X 0,Y 184.973,Z 328.211,A -85,B 0,C 180,E1 -23347.435,E2 -23347.435} C_VEL
LIN {X 0,Y 185.775,Z 326.23,A -85,B 0,C 180,E1 -23347.929,E2 -23347.929} C_VEL
LIN {X 0,Y 185.408,Z 317.648,A -85,B 0,C 180,E1 -23350.701,E2 -23350.701} C_VEL
LIN {X 0,Y 184.02,Z 308.768,A -85,B 0,C 180,E1 -23353.477,E2 -23353.477} C_VEL
LIN {X 0,Y 181.929,Z 300.901,A -85,B 0,C 180,E1 -23355.944,E2 -23355.944} C_VEL
LIN {X 0,Y 178.572,Z 292.631,A -85,B 0,C 180,E1 -23358.759,E2 -23358.759} C_VEL
LIN {X 0,Y 173.813,Z 283.193,A -85,B 0,C 180,E1 -23362.205,E2 -23362.205} C_VEL
LIN {X 0,Y 171.438,Z 279.288,A -85,B 0,C 180,E1 -23363.802,E2 -23363.802} C_VEL
LIN {X 0,Y 168.498,Z 274.945,A -85,B 0,C 180,E1 -23365.723,E2 -23365.723} C_VEL
LIN {X 0,Y 167.814,Z 273.654,A -85,B 0,C 180,E1 -23366.212,E2 -23366.212} C_VEL
LIN {X 0,Y 165.527,Z 271.182,A -85,B 0,C 180,E1 -23367.636,E2 -23367.636} C_VEL
LIN {X 0,Y 164.476,Z 268.583,A -85,B 0,C 180,E1 -23368.565,E2 -23368.565} C_VEL
LIN {X 0,Y 164.335,Z 268.008,A -85,B 0,C 180,E1 -23371.937,E2 -23371.937} C_VEL
LIN {X 0,Y 164.408,Z 268.006,A -85,B 0,C 180,E1 -23374.692,E2 -23374.692} C_VEL
LIN {X 0,Y 164.475,Z 267.996,A -85,B 0,C 180,E1 -23380.049,E2 -23380.049} C_VEL
LIN {X 0,Y 164.526,Z 267.992,A -85,B 0,C 180,E1 -23385.149,E2 -23385.149} C_VEL
LIN {X 0,Y 164.843,Z 267.951,A -85,B 0,C 180,E1 -23390.181,E2 -23390.181} C_VEL
LIN {X 0,Y 164.776,Z 267.959,A -85,B 0,C 180,E1 -23395.106,E2 -23395.106} C_VEL
LIN {X 0,Y 165.284,Z 267.896,A -85,B 0,C 180,E1 -23400,E2 -23400} C_VEL
LIN {X 0,Y 164.768,Z 267.959,A -85,B 0,C 180,E1 -23404.893,E2 -23404.893} C_VEL
LIN {X 0,Y 164.865,Z 268.032,A -85,B 0,C 180,E1 -23409.818,E2 -23409.818} C_VEL
LIN {X 0,Y 164.783,Z 269.451,A -85,B 0,C 180,E1 -23414.827,E2 -23414.827} C_VEL
LIN {X 0,Y 165.07,Z 271.408,A -85,B 0,C 180,E1 -23420.512,E2 -23420.512} C_VEL
LIN {X 0,Y 165.476,Z 274.097,A -85,B 0,C 180,E1 -23426.896,E2 -23426.896} C_VEL
LIN {X 0,Y 165.875,Z 276.641,A -85,B 0,C 180,E1 -23432.079,E2 -23432.079} C_VEL
LIN {X 0,Y 166.263,Z 279.241,A -85,B 0,C 180,E1 -23436.738,E2 -23436.738} C_VEL
LIN {X 0,Y 167.496,Z 282.555,A -85,B 0,C 180,E1 -23437.666,E2 -23437.666} C_VEL
LIN {X 0,Y 169.861,Z 285.638,A -85,B 0,C 180,E1 -23439.069,E2 -23439.069} C_VEL
